LIN {X 0,Y 93.573,Z 328.829,A -85,B 0,C 180,E1 -26788.279,E2 -26788.279} C_VEL
LIN {X 0,Y 93.645,Z 328.819,A -85,B 0,C 180,E1 -26794.239,E2 -26794.239} C_VEL
LIN {X 0,Y 93.653,Z 328.813,A -85,B 0,C 180,E1 -26797.96,E2 -26797.96} C_VEL
LIN {X 0,Y 94.018,Z 328.769,A -85,B 0,C 180,E1 -26807.039,E2 -26807.039} C_VEL
LIN {X 0,Y 94.131,Z 328.757,A -85,B 0,C 180,E1 -26811.41,E2 -26811.41} C_VEL
LIN {X 0,Y 94.763,Z 328.678,A -85,B 0,C 180,E1 -26819.998,E2 -26819.998} C_VEL
LIN {X 0,Y 94.13,Z 328.757,A -85,B 0,C 180,E1 -26828.586,E2 -26828.586} C_VEL
LIN {X 0,Y 93.956,Z 328.78,A -85,B 0,C 180,E1 -26833.486,E2 -26833.486} C_VEL
LIN {X 0,Y 93.653,Z 328.819,A -85,B 0,C 180,E1 -26842.035,E2 -26842.035} C_VEL
LIN {X 0,Y 93.601,Z 328.819,A -85,B 0,C 180,E1 -26846.774,E2 -26846.774} C_VEL
LIN {X 0,Y 93.584,Z 328.823,A -85,B 0,C 180,E1 -26854.298,E2 -26854.298} C_VEL
LIN {X 0,Y 93.537,Z 328.83,A -85,B 0,C 180,E1 -26862.546,E2 -26862.546} C_VEL
LIN {X 0,Y 93.555,Z 328.831,A -85,B 0,C 180,E1 -26868.692,E2 -26868.692} C_VEL
LIN {X 0,Y 93.602,Z 328.824,A -85,B 0,C 180,E1 -26875.679,E2 -26875.679} C_VEL
LIN {X 0,Y 93.669,Z 328.816,A -85,B 0,C 180,E1 -26884.201,E2 -26884.201} C_VEL
LIN {X 0,Y 93.693,Z 328.81,A -85,B 0,C 180,E1 -26887.967,E2 -26887.967} C_VEL
LIN {X 0,Y 94.082,Z 328.759,A -85,B 0,C 180,E1 -26897.044,E2 -26897.044} C_VEL
LIN {X 0,Y 94.207,Z 328.75,A -85,B 0,C 180,E1 -26901.413,E2 -26901.413} C_VEL
LIN {X 0,Y 94.794,Z 328.676,A -85,B 0,C 180,E1 -26909.993,E2 -26909.993} C_VEL
LIN {X 0,Y 94.21,Z 328.751,A -85,B 0,C 180,E1 -26918.573,E2 -26918.573} C_VEL
LIN {X 0,Y 94.181,Z 328.767,A -85,B 0,C 180,E1 -26921.834,E2 -26921.834} C_VEL
LIN {X 0,Y 95.166,Z 331.672,A -85,B 0,C 180,E1 -26922.521,E2 -26922.521} C_VEL
LIN {X 0,Y 101.569,Z 346.523,A -85,B 0,C 180,E1 -26926.174,E2 -26926.174} C_VEL
LIN {X 0,Y 109.633,Z 368.31,A -85,B 0,C 180,E1 -26930.466,E2 -26930.466} C_VEL
LIN {X 0,Y 110.536,Z 370.99,A -85,B 0,C 180,E1 -26930.925,E2 -26930.925} C_VEL
LIN {X 0,Y 105.93,Z 421.379,A -85,B 0,C 180,E1 -26935.46,E2 -26935.46} C_VEL
LIN {X 0,Y 104.057,Z 435.818,A -85,B 0,C 180,E1 -26937.573,E2 -26937.573} C_VEL
LIN {X 0,Y 101.762,Z 448.826,A -85,B 0,C 180,E1 -26940.316,E2 -26940.316} C_VEL
LIN {X 0,Y 99.25,Z 461.551,A -85,B 0,C 180,E1 -26943.946,E2 -26943.946} C_VEL
LIN {X 0,Y 96.668,Z 473.501,A -85,B 0,C 180,E1 -26948.496,E2 -26948.496} C_VEL
LIN {X 0,Y 94.521,Z 483.813,A -85,B 0,C 180,E1 -26953.539,E2 -26953.539} C_VEL
LIN {X 0,Y 92.739,Z 493.445,A -85,B 0,C 180,E1 -26959.62,E2 -26959.62} C_VEL
LIN {X 0,Y 91.805,Z 500.292,A -85,B 0,C 180,E1 -26964.963,E2 -26964.963} C_VEL
LIN {X 0,Y 91.274,Z 506.901,A -85,B 0,C 180,E1 -26971.276,E2 -26971.276} C_VEL
LIN {X 0,Y 91.876,Z 514.034,A -85,B 0,C 180,E1 -26979.868,E2 -26979.868} C_VEL
LIN {X 0,Y 93.831,Z 518.658,A -85,B 0,C 180,E1 -26987.017,E2 -26987.017} C_VEL
LIN {X 0,Y 95.951,Z 521.091,A -85,B 0,C 180,E1 -26991.578,E2 -26991.578} C_VEL
LIN {X 0,Y 98.609,Z 523.092,A -85,B 0,C 180,E1 -26996.015,E2 -26996.015} C_VEL
LIN {X 0,Y 101.749,Z 524.592,A -85,B 0,C 180,E1 -27000.002,E2 -27000.002} C_VEL
LIN {X 0,Y 105.656,Z 525.69,A -85,B 0,C 180,E1 -27004.008,E2 -27004.008} C_VEL
LIN {X 0,Y 109.634,Z 526.281,A -85,B 0,C 180,E1 -27007.368,E2 -27007.368} C_VEL
LIN {X 0,Y 114.426,Z 526.503,A -85,B 0,C 180,E1 -27010.73,E2 -27010.73} C_VEL
LIN {X 0,Y 119.307,Z 526.284,A -85,B 0,C 180,E1 -27013.63,E2 -27013.63} C_VEL
LIN {X 0,Y 124.666,Z 525.596,A -85,B 0,C 180,E1 -27016.374,E2 -27016.374} C_VEL
LIN {X 0,Y 135.294,Z 523.2,A -85,B 0,C 180,E1 -27020.795,E2 -27020.795} C_VEL
LIN {X 0,Y 146.652,Z 519.189,A -85,B 0,C 180,E1 -27024.444,E2 -27024.444} C_VEL
LIN {X 0,Y 158.313,Z 513.62,A -85,B 0,C 180,E1 -27027.414,E2 -27027.414} C_VEL
LIN {X 0,Y 167.136,Z 508.313,A -85,B 0,C 180,E1 -27029.296,E2 -27029.296} C_VEL
LIN {X 0,Y 165.242,Z 509.715,A -85,B 0,C 180,E1 -27030.279,E2 -27030.279} C_VEL
LIN {X 0,Y 154.143,Z 516.659,A -85,B 0,C 180,E1 -27032.507,E2 -27032.507} C_VEL
LIN {X 0,Y 145.218,Z 521.23,A -85,B 0,C 180,E1 -27034.657,E2 -27034.657} C_VEL
LIN {X 0,Y 133.848,Z 525.943,A -85,B 0,C 180,E1 -27038.053,E2 -27038.053} C_VEL
LIN {X 0,Y 123.437,Z 529.163,A -85,B 0,C 180,E1 -27042.268,E2 -27042.268} C_VEL
LIN {X 0,Y 114.003,Z 531.067,A -85,B 0,C 180,E1 -27047.316,E2 -27047.316} C_VEL
LIN {X 0,Y 106.022,Z 531.693,A -85,B 0,C 180,E1 -27053.386,E2 -27053.386} C_VEL
LIN {X 0,Y 99.465,Z 530.999,A -85,B 0,C 180,E1 -27060.367,E2 -27060.367} C_VEL
LIN {X 0,Y 94.915,Z 528.991,A -85,B 0,C 180,E1 -27068.28,E2 -27068.28} C_VEL
LIN {X 0,Y 92.801,Z 525.673,A -85,B 0,C 180,E1 -27076.876,E2 -27076.876} C_VEL
LIN {X 0,Y 92.558,Z 522.492,A -85,B 0,C 180,E1 -27082.906,E2 -27082.906} C_VEL
LIN {X 0,Y 92.895,Z 519.232,A -85,B 0,C 180,E1 -27087.839,E2 -27087.839} C_VEL
LIN {X 0,Y 92.777,Z 514.534,A -85,B 0,C 180,E1 -27093.264,E2 -27093.264} C_VEL
LIN {X 0,Y 92.839,Z 508.649,A -85,B 0,C 180,E1 -27098.714,E2 -27098.714} C_VEL
LIN {X 0,Y 93.733,Z 499.874,A -85,B 0,C 180,E1 -27105.22,E2 -27105.22} C_VEL
LIN {X 0,Y 95.279,Z 490.866,A -85,B 0,C 180,E1 -27110.515,E2 -27110.515} C_VEL
LIN {X 0,Y 97.615,Z 479.729,A -85,B 0,C 180,E1 -27115.598,E2 -27115.598} C_VEL
LIN {X 0,Y 99.953,Z 468.688,A -85,B 0,C 180,E1 -27119.489,E2 -27119.489} C_VEL
LIN {X 0,Y 102.558,Z 455.448,A -85,B 0,C 180,E1 -27122.955,E2 -27122.955} C_VEL
LIN {X 0,Y 104.664,Z 442.605,A -85,B 0,C 180,E1 -27125.394,E2 -27125.394} C_VEL
LIN {X 0,Y 106.08,Z 430.388,A -85,B 0,C 180,E1 -27127.008,E2 -27127.008} C_VEL
LIN {X 0,Y 109.326,Z 392.754,A -85,B 0,C 180,E1 -27130.449,E2 -27130.449} C_VEL
LIN {X 0,Y 107.869,Z 369.994,A -85,B 0,C 180,E1 -27133.101,E2 -27133.101} C_VEL
LIN {X 0,Y 107.342,Z 367.864,A -85,B 0,C 180,E1 -27133.437,E2 -27133.437} C_VEL
LIN {X 0,Y 105.36,Z 362.63,A -85,B 0,C 180,E1 -27134.438,E2 -27134.438} C_VEL
LIN {X 0,Y 100.496,Z 354.863,A -85,B 0,C 180,E1 -27136.508,E2 -27136.508} C_VEL
LIN {X 0,Y 96.186,Z 348.926,A -85,B 0,C 180,E1 -27138.421,E2 -27138.421} C_VEL
LIN {X 0,Y 92.4,Z 342.627,A -85,B 0,C 180,E1 -27140.358,E2 -27140.358} C_VEL
LIN {X 0,Y 87.501,Z 332.578,A -85,B 0,C 180,E1 -27143.394,E2 -27143.394} C_VEL
LIN {X 0,Y 86.506,Z 329.708,A -85,B 0,C 180,E1 -27144.339,E2 -27144.339} C_VEL
LIN {X 0,Y 86.567,Z 329.702,A -85,B 0,C 180,E1 -27153.263,E2 -27153.263} C_VEL
LIN {X 0,Y 86.598,Z 329.698,A -85,B 0,C 180,E1 -27161.055,E2 -27161.055} C_VEL
LIN {X 0,Y 86.861,Z 329.658,A -85,B 0,C 180,E1 -27166.158,E2 -27166.158} C_VEL
LIN {X 0,Y 87.026,Z 329.644,A -85,B 0,C 180,E1 -27170.703,E2 -27170.703} C_VEL
LIN {X 0,Y 87.693,Z 329.559,A -85,B 0,C 180,E1 -27179.998,E2 -27179.998} C_VEL
LIN {X 0,Y 87.024,Z 329.639,A -85,B 0,C 180,E1 -27189.293,E2 -27189.293} C_VEL
LIN {X 0,Y 86.86,Z 329.666,A -85,B 0,C 180,E1 -27194.046,E2 -27194.046} C_VEL
LIN {X 0,Y 86.597,Z 329.69,A -85,B 0,C 180,E1 -27198.941,E2 -27198.941} C_VEL
LIN {X 0,Y 86.566,Z 329.695,A -85,B 0,C 180,E1 -27206.736,E2 -27206.736} C_VEL
LIN {X 0,Y 86.504,Z 329.702,A -85,B 0,C 180,E1 -27215.659,E2 -27215.659} C_VEL
LIN {X 0,Y 86.48,Z 329.708,A -85,B 0,C 180,E1 -27222.991,E2 -27222.991} C_VEL
LIN {X 0,Y 86.475,Z 329.713,A -85,B 0,C 180,E1 -27229.44,E2 -27229.44} C_VEL
LIN {X 0,Y 86.547,Z 329.703,A -85,B 0,C 180,E1 -27235.354,E2 -27235.354} C_VEL
LIN {X 0,Y 86.584,Z 329.697,A -85,B 0,C 180,E1 -27243.231,E2 -27243.231} C_VEL
LIN {X 0,Y 86.646,Z 329.687,A -85,B 0,C 180,E1 -27251.062,E2 -27251.062} C_VEL
LIN {X 0,Y 86.95,Z 329.651,A -85,B 0,C 180,E1 -27255.961,E2 -27255.961} C_VEL
LIN {X 0,Y 87.111,Z 329.633,A -85,B 0,C 180,E1 -27260.708,E2 -27260.708} C_VEL
LIN {X 0,Y 87.722,Z 329.558,A -85,B 0,C 180,E1 -27269.993,E2 -27269.993} C_VEL
LIN {X 0,Y 87.135,Z 329.63,A -85,B 0,C 180,E1 -27279.421,E2 -27279.421} C_VEL
LIN {X 0,Y 88.182,Z 332.606,A -85,B 0,C 180,E1 -27280.249,E2 -27280.249} C_VEL
LIN {X 0,Y 94.846,Z 347.726,A -85,B 0,C 180,E1 -27284.444,E2 -27284.444} C_VEL
LIN {X 0,Y 102.434,Z 368.321,A -85,B 0,C 180,E1 -27288.89,E2 -27288.89} C_VEL
LIN {X 0,Y 103.782,Z 372.236,A -85,B 0,C 180,E1 -27289.638,E2 -27289.638} C_VEL
LIN {X 0,Y 99.129,Z 421.425,A -85,B 0,C 180,E1 -27294.314,E2 -27294.314} C_VEL
LIN {X 0,Y 97.199,Z 435.818,A -85,B 0,C 180,E1 -27296.53,E2 -27296.53} C_VEL
LIN {X 0,Y 94.953,Z 448.117,A -85,B 0,C 180,E1 -27299.226,E2 -27299.226} C_VEL
LIN {X 0,Y 92.302,Z 461.049,A -85,B 0,C 180,E1 -27303.121,E2 -27303.121} C_VEL
LIN {X 0,Y 89.803,Z 472.245,A -85,B 0,C 180,E1 -27307.595,E2 -27307.595} C_VEL
LIN {X 0,Y 87.602,Z 482.61,A -85,B 0,C 180,E1 -27312.944,E2 -27312.944} C_VEL
LIN {X 0,Y 85.789,Z 491.966,A -85,B 0,C 180,E1 -27319.055,E2 -27319.055} C_VEL
LIN {X 0,Y 84.854,Z 498.799,A -85,B 0,C 180,E1 -27324.568,E2 -27324.568} C_VEL
LIN {X 0,Y 84.283,Z 505.708,A -85,B 0,C 180,E1 -27331.352,E2 -27331.352} C_VEL
LIN {X 0,Y 84.613,Z 511.599,A -85,B 0,C 180,E1 -27338.541,E2 -27338.541} C_VEL
LIN {X 0,Y 86.562,Z 517.223,A -85,B 0,C 180,E1 -27346.919,E2 -27346.919} C_VEL
LIN {X 0,Y 90.737,Z 521.822,A -85,B 0,C 180,E1 -27355.56,E2 -27355.56} C_VEL
LIN {X 0,Y 93.852,Z 523.72,A -85,B 0,C 180,E1 -27360.002,E2 -27360.002} C_VEL
LIN {X 0,Y 98.798,Z 525.543,A -85,B 0,C 180,E1 -27365.331,E2 -27365.331} C_VEL
LIN {X 0,Y 107.894,Z 526.949,A -85,B 0,C 180,E1 -27372.349,E2 -27372.349} C_VEL
LIN {X 0,Y 118.23,Z 526.65,A -85,B 0,C 180,E1 -27378.029,E2 -27378.029} C_VEL
LIN {X 0,Y 129.371,Z 524.824,A -85,B 0,C 180,E1 -27382.582,E2 -27382.582} C_VEL
LIN {X 0,Y 135.32,Z 523.307,A -85,B 0,C 180,E1 -27384.552,E2 -27384.552} C_VEL
LIN {X 0,Y 145.313,Z 519.918,A -85,B 0,C 180,E1 -27387.354,E2 -27387.354} C_VEL
LIN {X 0,Y 152.834,Z 516.661,A -85,B 0,C 180,E1 -27389.127,E2 -27389.127} C_VEL
LIN {X 0,Y 153.61,Z 516.346,A -85,B 0,C 180,E1 -27389.642,E2 -27389.642} C_VEL
LIN {X 0,Y 144.329,Z 520.911,A -85,B 0,C 180,E1 -27391.572,E2 -27391.572} C_VEL
LIN {X 0,Y 135.409,Z 524.497,A -85,B 0,C 180,E1 -27393.874,E2 -27393.874} C_VEL
LIN {X 0,Y 129.616,Z 526.446,A -85,B 0,C 180,E1 -27395.595,E2 -27395.595} C_VEL
LIN {X 0,Y 118.788,Z 529.296,A -85,B 0,C 180,E1 -27399.739,E2 -27399.739} C_VEL
LIN {X 0,Y 108.887,Z 530.811,A -85,B 0,C 180,E1 -27404.781,E2 -27404.781} C_VEL
LIN {X 0,Y 100.416,Z 531.081,A -85,B 0,C 180,E1 -27410.97,E2 -27410.97} C_VEL
LIN {X 0,Y 93.38,Z 530.082,A -85,B 0,C 180,E1 -27418.22,E2 -27418.22} C_VEL
LIN {X 0,Y 88.425,Z 527.802,A -85,B 0,C 180,E1 -27426.595,E2 -27426.595} C_VEL
LIN {X 0,Y 86.034,Z 524.174,A -85,B 0,C 180,E1 -27435.823,E2 -27435.823} C_VEL
LIN {X 0,Y 85.757,Z 520.047,A -85,B 0,C 180,E1 -27443.597,E2 -27443.597} C_VEL
LIN {X 0,Y 86.024,Z 517.323,A -85,B 0,C 180,E1 -27447.667,E2 -27447.667} C_VEL
LIN {X 0,Y 85.863,Z 512.343,A -85,B 0,C 180,E1 -27453.527,E2 -27453.527} C_VEL
LIN {X 0,Y 86.057,Z 504.633,A -85,B 0,C 180,E1 -27460.654,E2 -27460.654} C_VEL
LIN {X 0,Y 87.377,Z 495.19,A -85,B 0,C 180,E1 -27467.561,E2 -27467.561} C_VEL
LIN {X 0,Y 89.255,Z 485.216,A -85,B 0,C 180,E1 -27473.191,E2 -27473.191} C_VEL
LIN {X 0,Y 91.665,Z 474.119,A -85,B 0,C 180,E1 -27478.014,E2 -27478.014} C_VEL
LIN {X 0,Y 93.944,Z 463.458,A -85,B 0,C 180,E1 -27481.583,E2 -27481.583} C_VEL
LIN {X 0,Y 96.379,Z 450.858,A -85,B 0,C 180,E1 -27484.733,E2 -27484.733} C_VEL
LIN {X 0,Y 98.532,Z 437.173,A -85,B 0,C 180,E1 -27487.165,E2 -27487.165} C_VEL
LIN {X 0,Y 100.132,Z 420.928,A -85,B 0,C 180,E1 -27489.016,E2 -27489.016} C_VEL
LIN {X 0,Y 102.571,Z 392.894,A -85,B 0,C 180,E1 -27491.696,E2 -27491.696} C_VEL
LIN {X 0,Y 101.351,Z 371.639,A -85,B 0,C 180,E1 -27494.346,E2 -27494.346} C_VEL
LIN {X 0,Y 95.522,Z 351.056,A -85,B 0,C 180,E1 -27498.356,E2 -27498.356} C_VEL
LIN {X 0,Y 93.12,Z 344.081,A -85,B 0,C 180,E1 -27499.948,E2 -27499.948} C_VEL
LIN {X 0,Y 92.4,Z 342.627,A -85,B 0,C 180,E1 -27500.358,E2 -27500.358} C_VEL
LIN {X 0,Y 89.675,Z 338.423,A -85,B 0,C 180,E1 -27502.024,E2 -27502.024} C_VEL
LIN {X 0,Y 86.516,Z 335.212,A -85,B 0,C 180,E1 -27504.303,E2 -27504.303} C_VEL
LIN {X 0,Y 84.439,Z 333.568,A -85,B 0,C 180,E1 -27506.148,E2 -27506.148} C_VEL
LIN {X 0,Y 81.696,Z 331.776,A -85,B 0,C 180,E1 -27509.405,E2 -27509.405} C_VEL
LIN {X 0,Y 79.855,Z 330.78,A -85,B 0,C 180,E1 -27513.182,E2 -27513.182} C_VEL
LIN {X 0,Y 79.409,Z 330.581,A -85,B 0,C 180,E1 -27515.896,E2 -27515.896} C_VEL
LIN {X 0,Y 79.69,Z 330.551,A -85,B 0,C 180,E1 -27524.656,E2 -27524.656} C_VEL
LIN {X 0,Y 79.91,Z 330.531,A -85,B 0,C 180,E1 -27529.867,E2 -27529.867} C_VEL
LIN {X 0,Y 80.622,Z 330.44,A -85,B 0,C 180,E1 -27539.998,E2 -27539.998} C_VEL
LIN {X 0,Y 79.909,Z 330.523,A -85,B 0,C 180,E1 -27550.128,E2 -27550.128} C_VEL
LIN {X 0,Y 79.688,Z 330.559,A -85,B 0,C 180,E1 -27555.339,E2 -27555.339} C_VEL
LIN {X 0,Y 79.476,Z 330.581,A -85,B 0,C 180,E1 -27560.712,E2 -27560.712} C_VEL
LIN {X 0,Y 79.468,Z 330.578,A -85,B 0,C 180,E1 -27567.818,E2 -27567.818} C_VEL
LIN {X 0,Y 79.372,Z 330.598,A -85,B 0,C 180,E1 -27572.088,E2 -27572.088} C_VEL
LIN {X 0,Y 79.365,Z 330.597,A -85,B 0,C 180,E1 -27578.303,E2 -27578.303} C_VEL
LIN {X 0,Y 79.412,Z 330.586,A -85,B 0,C 180,E1 -27585.069,E2 -27585.069} C_VEL
LIN {X 0,Y 79.399,Z 330.586,A -85,B 0,C 180,E1 -27592.806,E2 -27592.806} C_VEL
LIN {X 0,Y 79.386,Z 330.596,A -85,B 0,C 180,E1 -27597.909,E2 -27597.909} C_VEL
LIN {X 0,Y 79.525,Z 330.577,A -85,B 0,C 180,E1 -27603.77,E2 -27603.77} C_VEL
LIN {X 0,Y 79.513,Z 330.572,A -85,B 0,C 180,E1 -27609.289,E2 -27609.289} C_VEL
LIN {X 0,Y 79.838,Z 330.538,A -85,B 0,C 180,E1 -27615.526,E2 -27615.526} C_VEL
LIN {X 0,Y 79.991,Z 330.518,A -85,B 0,C 180,E1 -27619.872,E2 -27619.872} C_VEL
LIN {X 0,Y 80.65,Z 330.439,A -85,B 0,C 180,E1 -27629.992,E2 -27629.992} C_VEL
LIN {X 0,Y 80.082,Z 330.514,A -85,B 0,C 180,E1 -27636.606,E2 -27636.606} C_VEL
LIN {X 0,Y 81.156,Z 333.469,A -85,B 0,C 180,E1 -27637.533,E2 -27637.533} C_VEL
LIN {X 0,Y 84.237,Z 339.738,A -85,B 0,C 180,E1 -27639.747,E2 -27639.747} C_VEL
LIN {X 0,Y 89.836,Z 353.407,A -85,B 0,C 180,E1 -27643.654,E2 -27643.654} C_VEL
LIN {X 0,Y 96.539,Z 371.954,A -85,B 0,C 180,E1 -27647.861,E2 -27647.861} C_VEL
LIN {X 0,Y 97.091,Z 374.405,A -85,B 0,C 180,E1 -27648.287,E2 -27648.287} C_VEL
LIN {X 0,Y 92.273,Z 422.261,A -85,B 0,C 180,E1 -27653.172,E2 -27653.172} C_VEL
LIN {X 0,Y 90.132,Z 436.987,A -85,B 0,C 180,E1 -27655.639,E2 -27655.639} C_VEL
LIN {X 0,Y 87.69,Z 449.666,A -85,B 0,C 180,E1 -27658.731,E2 -27658.731} C_VEL
LIN {X 0,Y 84.893,Z 462.653,A -85,B 0,C 180,E1 -27663.053,E2 -27663.053} C_VEL
LIN {X 0,Y 82.253,Z 474.252,A -85,B 0,C 180,E1 -27668.264,E2 -27668.264} C_VEL
LIN {X 0,Y 80.132,Z 483.916,A -85,B 0,C 180,E1 -27673.837,E2 -27673.837} C_VEL
LIN {X 0,Y 78.624,Z 491.944,A -85,B 0,C 180,E1 -27679.608,E2 -27679.608} C_VEL
LIN {X 0,Y 77.569,Z 500.264,A -85,B 0,C 180,E1 -27687.073,E2 -27687.073} C_VEL
LIN {X 0,Y 77.327,Z 507.531,A -85,B 0,C 180,E1 -27695.317,E2 -27695.317} C_VEL
LIN {X 0,Y 78.687,Z 514.056,A -85,B 0,C 180,E1 -27704.46,E2 -27704.46} C_VEL
LIN {X 0,Y 81.576,Z 518.831,A -85,B 0,C 180,E1 -27712.577,E2 -27712.577} C_VEL
LIN {X 0,Y 85.984,Z 522.477,A -85,B 0,C 180,E1 -27720.002,E2 -27720.002} C_VEL
LIN {X 0,Y 92.002,Z 525.211,A -85,B 0,C 180,E1 -27726.858,E2 -27726.858} C_VEL
LIN {X 0,Y 101.475,Z 527.183,A -85,B 0,C 180,E1 -27734.208,E2 -27734.208} C_VEL
LIN {X 0,Y 112.153,Z 527.456,A -85,B 0,C 180,E1 -27739.987,E2 -27739.987} C_VEL
LIN {X 0,Y 123.603,Z 526.25,A -85,B 0,C 180,E1 -27744.554,E2 -27744.554} C_VEL
LIN {X 0,Y 135.477,Z 523.546,A -85,B 0,C 180,E1 -27748.149,E2 -27748.149} C_VEL
LIN {X 0,Y 138.821,Z 522.561,A -85,B 0,C 180,E1 -27749.023,E2 -27749.023} C_VEL
LIN {X 0,Y 137.697,Z 523.035,A -85,B 0,C 180,E1 -27749.831,E2 -27749.831} C_VEL
LIN {X 0,Y 125.623,Z 526.855,A -85,B 0,C 180,E1 -27752.965,E2 -27752.965} C_VEL
LIN {X 0,Y 114.378,Z 529.299,A -85,B 0,C 180,E1 -27757.003,E2 -27757.003} C_VEL
LIN {X 0,Y 104.02,Z 530.489,A -85,B 0,C 180,E1 -27762.01,E2 -27762.01} C_VEL
LIN {X 0,Y 95.011,Z 530.427,A -85,B 0,C 180,E1 -27768.276,E2 -27768.276} C_VEL
LIN {X 0,Y 87.46,Z 529.073,A -85,B 0,C 180,E1 -27775.784,E2 -27775.784} C_VEL
LIN {X 0,Y 82.043,Z 526.479,A -85,B 0,C 180,E1 -27784.651,E2 -27784.651} C_VEL
LIN {X 0,Y 79.333,Z 522.546,A -85,B 0,C 180,E1 -27794.597,E2 -27794.597} C_VEL
LIN {X 0,Y 78.937,Z 518.578,A -85,B 0,C 180,E1 -27802.334,E2 -27802.334} C_VEL
LIN {X 0,Y 79.172,Z 515.331,A -85,B 0,C 180,E1 -27807.465,E2 -27807.465} C_VEL
LIN {X 0,Y 78.966,Z 509.994,A -85,B 0,C 180,E1 -27813.835,E2 -27813.835} C_VEL
LIN {X 0,Y 79.247,Z 501.612,A -85,B 0,C 180,E1 -27821.793,E2 -27821.793} C_VEL
LIN {X 0,Y 80.764,Z 491.781,A -85,B 0,C 180,E1 -27829.052,E2 -27829.052} C_VEL
LIN {X 0,Y 82.905,Z 481.221,A -85,B 0,C 180,E1 -27835.084,E2 -27835.084} C_VEL
LIN {X 0,Y 85.595,Z 469.314,A -85,B 0,C 180,E1 -27840.198,E2 -27840.198} C_VEL
LIN {X 0,Y 88.112,Z 457.694,A -85,B 0,C 180,E1 -27843.946,E2 -27843.946} C_VEL
LIN {X 0,Y 90.533,Z 444.586,A -85,B 0,C 180,E1 -27846.991,E2 -27846.991} C_VEL
LIN {X 0,Y 92.221,Z 432.548,A -85,B 0,C 180,E1 -27848.96,E2 -27848.96} C_VEL
LIN {X 0,Y 95.931,Z 394.052,A -85,B 0,C 180,E1 -27852.985,E2 -27852.985} C_VEL
LIN {X 0,Y 94.901,Z 373.415,A -85,B 0,C 180,E1 -27855.751,E2 -27855.751} C_VEL
LIN {X 0,Y 89.374,Z 353.596,A -85,B 0,C 180,E1 -27859.863,E2 -27859.863} C_VEL
LIN {X 0,Y 87.144,Z 347.089,A -85,B 0,C 180,E1 -27861.494,E2 -27861.494} C_VEL
LIN {X 0,Y 81.935,Z 336.258,A -85,B 0,C 180,E1 -27865.085,E2 -27865.085} C_VEL
LIN {X 0,Y 79.562,Z 331.488,A -85,B 0,C 180,E1 -27866.865,E2 -27866.865} C_VEL
LIN {X 0,Y 79.395,Z 330.594,A -85,B 0,C 180,E1 -27867.165,E2 -27867.165} C_VEL
LIN {X 0,Y 79.508,Z 330.58,A -85,B 0,C 180,E1 -27873.768,E2 -27873.768} C_VEL
LIN {X 0,Y 79.409,Z 330.581,A -85,B 0,C 180,E1 -27875.896,E2 -27875.896} C_VEL
LIN {X 0,Y 78.681,Z 330.683,A -85,B 0,C 180,E1 -27880.134,E2 -27880.134} C_VEL
LIN {X 0,Y 77.128,Z 330.878,A -85,B 0,C 180,E1 -27884.358,E2 -27884.358} C_VEL
LIN {X 0,Y 73.356,Z 331.346,A -85,B 0,C 180,E1 -27896.354,E2 -27896.354} C_VEL
LIN {X 0,Y 73.472,Z 331.326,A -85,B 0,C 180,E1 -27899.511,E2 -27899.511} C_VEL
LIN {X 0,Y 72.916,Z 331.395,A -85,B 0,C 180,E1 -27906.381,E2 -27906.381} C_VEL
LIN {X 0,Y 72.809,Z 331.407,A -85,B 0,C 180,E1 -27911.128,E2 -27911.128} C_VEL
LIN {X 0,Y 72.506,Z 331.45,A -85,B 0,C 180,E1 -27916.902,E2 -27916.902} C_VEL
LIN {X 0,Y 72.367,Z 331.47,A -85,B 0,C 180,E1 -27922.856,E2 -27922.856} C_VEL
LIN {X 0,Y 72.36,Z 331.466,A -85,B 0,C 180,E1 -27929.05,E2 -27929.05} C_VEL
LIN {X 0,Y 72.292,Z 331.472,A -85,B 0,C 180,E1 -27935.68,E2 -27935.68} C_VEL
LIN {X 0,Y 72.261,Z 331.478,A -85,B 0,C 180,E1 -27942.903,E2 -27942.903} C_VEL
LIN {X 0,Y 72.306,Z 331.474,A -85,B 0,C 180,E1 -27951.036,E2 -27951.036} C_VEL
LIN {X 0,Y 72.304,Z 331.473,A -85,B 0,C 180,E1 -27954.317,E2 -27954.317} C_VEL
LIN {X 0,Y 72.376,Z 331.461,A -85,B 0,C 180,E1 -27960.946,E2 -27960.946} C_VEL
LIN {X 0,Y 72.394,Z 331.465,A -85,B 0,C 180,E1 -27967.143,E2 -27967.143} C_VEL
LIN {X 0,Y 72.755,Z 331.421,A -85,B 0,C 180,E1 -27975.002,E2 -27975.002} C_VEL
LIN {X 0,Y 72.878,Z 331.4,A -85,B 0,C 180,E1 -27978.872,E2 -27978.872} C_VEL
LIN {X 0,Y 73.577,Z 331.32,A -85,B 0,C 180,E1 -27989.991,E2 -27989.991} C_VEL
LIN {X 0,Y 73.219,Z 331.359,A -85,B 0,C 180,E1 -27993.258,E2 -27993.258} C_VEL
LIN {X 0,Y 74.182,Z 334.307,A -85,B 0,C 180,E1 -27994.406,E2 -27994.406} C_VEL
LIN {X 0,Y 78.483,Z 342.94,A -85,B 0,C 180,E1 -27997.882,E2 -27997.882} C_VEL
LIN {X 0,Y 84.157,Z 357.131,A -85,B 0,C 180,E1 -28002.255,E2 -28002.255} C_VEL
LIN {X 0,Y 90.319,Z 374.686,A -85,B 0,C 180,E1 -28006.596,E2 -28006.596} C_VEL
LIN {X 0,Y 85.443,Z 422.933,A -85,B 0,C 180,E1 -28011.893,E2 -28011.893} C_VEL
LIN {X 0,Y 83.187,Z 437.447,A -85,B 0,C 180,E1 -28014.493,E2 -28014.493} C_VEL
LIN {X 0,Y 80.496,Z 450.947,A -85,B 0,C 180,E1 -28018.078,E2 -28018.078} C_VEL
LIN {X 0,Y 77.779,Z 462.885,A -85,B 0,C 180,E1 -28022.405,E2 -28022.405} C_VEL
LIN {X 0,Y 74.967,Z 474.83,A -85,B 0,C 180,E1 -28028.27,E2 -28028.27} C_VEL
LIN {X 0,Y 72.769,Z 484.728,A -85,B 0,C 180,E1 -28034.651,E2 -28034.651} C_VEL
LIN {X 0,Y 71.202,Z 493.839,A -85,B 0,C 180,E1 -28042.13,E2 -28042.13} C_VEL
LIN {X 0,Y 70.429,Z 501.536,A -85,B 0,C 180,E1 -28050.073,E2 -28050.073} C_VEL
LIN {X 0,Y 70.705,Z 508.983,A -85,B 0,C 180,E1 -28059.644,E2 -28059.644} C_VEL
LIN {X 0,Y 72.767,Z 514.871,A -85,B 0,C 180,E1 -28068.865,E2 -28068.865} C_VEL
LIN {X 0,Y 77.311,Z 520.21,A -85,B 0,C 180,E1 -28078.619,E2 -28078.619} C_VEL
LIN {X 0,Y 81.843,Z 523.141,A -85,B 0,C 180,E1 -28084.929,E2 -28084.929} C_VEL
LIN {X 0,Y 86.119,Z 524.977,A -85,B 0,C 180,E1 -28089.396,E2 -28089.396} C_VEL
LIN {X 0,Y 95.175,Z 527.199,A -85,B 0,C 180,E1 -28096.314,E2 -28096.314} C_VEL
LIN {X 0,Y 106.253,Z 528.059,A -85,B 0,C 180,E1 -28102.209,E2 -28102.209} C_VEL
LIN {X 0,Y 118.057,Z 527.436,A -85,B 0,C 180,E1 -28106.776,E2 -28106.776} C_VEL
LIN {X 0,Y 124.606,Z 526.461,A -85,B 0,C 180,E1 -28108.795,E2 -28108.795} C_VEL
LIN {X 0,Y 123.272,Z 526.883,A -85,B 0,C 180,E1 -28109.813,E2 -28109.813} C_VEL
LIN {X 0,Y 110.256,Z 529.223,A -85,B 0,C 180,E1 -28114.059,E2 -28114.059} C_VEL
LIN {X 0,Y 99.411,Z 530.023,A -85,B 0,C 180,E1 -28118.97,E2 -28118.97} C_VEL
LIN {X 0,Y 89.845,Z 529.619,A -85,B 0,C 180,E1 -28125.266,E2 -28125.266} C_VEL
LIN {X 0,Y 81.732,Z 527.988,A -85,B 0,C 180,E1 -28133.007,E2 -28133.007} C_VEL
LIN {X 0,Y 75.797,Z 525.061,A -85,B 0,C 180,E1 -28142.393,E2 -28142.393} C_VEL
LIN {X 0,Y 72.702,Z 520.826,A -85,B 0,C 180,E1 -28153.153,E2 -28153.153} C_VEL
LIN {X 0,Y 72.366,Z 514.983,A -85,B 0,C 180,E1 -28164.436,E2 -28164.436} C_VEL
LIN {X 0,Y 72.226,Z 511.047,A -85,B 0,C 180,E1 -28170.009,E2 -28170.009} C_VEL
LIN {X 0,Y 72.039,Z 504.91,A -85,B 0,C 180,E1 -28177.013,E2 -28177.013} C_VEL
LIN {X 0,Y 72.859,Z 495.797,A -85,B 0,C 180,E1 -28185.28,E2 -28185.28} C_VEL
LIN {X 0,Y 74.603,Z 486.121,A -85,B 0,C 180,E1 -28192.144,E2 -28192.144} C_VEL
LIN {X 0,Y 76.997,Z 475.592,A -85,B 0,C 180,E1 -28197.898,E2 -28197.898} C_VEL
LIN {X 0,Y 79.67,Z 463.896,A -85,B 0,C 180,E1 -28202.71,E2 -28202.71} C_VEL
LIN {X 0,Y 82.233,Z 451.901,A -85,B 0,C 180,E1 -28206.369,E2 -28206.369} C_VEL
LIN {X 0,Y 84.642,Z 438.246,A -85,B 0,C 180,E1 -28209.286,E2 -28209.286} C_VEL
LIN {X 0,Y 86.259,Z 424.458,A -85,B 0,C 180,E1 -28211.26,E2 -28211.26} C_VEL
LIN {X 0,Y 89.228,Z 393.764,A -85,B 0,C 180,E1 -28214.608,E2 -28214.608} C_VEL
LIN {X 0,Y 88.341,Z 374.688,A -85,B 0,C 180,E1 -28217.351,E2 -28217.351} C_VEL
LIN {X 0,Y 82.585,Z 353.674,A -85,B 0,C 180,E1 -28222.2,E2 -28222.2} C_VEL
LIN {X 0,Y 78.483,Z 343.957,A -85,B 0,C 180,E1 -28225.385,E2 -28225.385} C_VEL
LIN {X 0,Y 73.68,Z 334.843,A -85,B 0,C 180,E1 -28229.152,E2 -28229.152} C_VEL
LIN {X 0,Y 72.51,Z 332.392,A -85,B 0,C 180,E1 -28230.213,E2 -28230.213} C_VEL
LIN {X 0,Y 72.34,Z 331.473,A -85,B 0,C 180,E1 -28230.536,E2 -28230.536} C_VEL
LIN {X 0,Y 72.369,Z 331.462,A -85,B 0,C 180,E1 -28237.139,E2 -28237.139} C_VEL
LIN {X 0,Y 72.68,Z 331.423,A -85,B 0,C 180,E1 -28245.246,E2 -28245.246} C_VEL
LIN {X 0,Y 72.81,Z 331.415,A -85,B 0,C 180,E1 -28248.866,E2 -28248.866} C_VEL
LIN {X 0,Y 73.472,Z 331.326,A -85,B 0,C 180,E1 -28259.511,E2 -28259.511} C_VEL
LIN {X 0,Y 73.413,Z 331.347,A -85,B 0,C 180,E1 -28262.522,E2 -28262.522} C_VEL
LIN {X 0,Y 71.964,Z 331.527,A -85,B 0,C 180,E1 -28267.002,E2 -28267.002} C_VEL
LIN {X 0,Y 69.692,Z 331.796,A -85,B 0,C 180,E1 -28271.467,E2 -28271.467} C_VEL
LIN {X 0,Y 65.498,Z 332.324,A -85,B 0,C 180,E1 -28281.55,E2 -28281.55} C_VEL
LIN {X 0,Y 65.202,Z 332.356,A -85,B 0,C 180,E1 -28285.203,E2 -28285.203} C_VEL
LIN {X 0,Y 65.171,Z 332.366,A -85,B 0,C 180,E1 -28292.625,E2 -28292.625} C_VEL
LIN {X 0,Y 65.191,Z 332.364,A -85,B 0,C 180,E1 -28300.998,E2 -28300.998} C_VEL
LIN {X 0,Y 65.216,Z 332.36,A -85,B 0,C 180,E1 -28309.707,E2 -28309.707} C_VEL
LIN {X 0,Y 65.256,Z 332.351,A -85,B 0,C 180,E1 -28319.489,E2 -28319.489} C_VEL
LIN {X 0,Y 65.239,Z 332.358,A -85,B 0,C 180,E1 -28324.467,E2 -28324.467} C_VEL
LIN {X 0,Y 65.649,Z 332.307,A -85,B 0,C 180,E1 -28334.457,E2 -28334.457} C_VEL
LIN {X 0,Y 65.778,Z 332.283,A -85,B 0,C 180,E1 -28337.653,E2 -28337.653} C_VEL
LIN {X 0,Y 66.414,Z 332.32,A -85,B 0,C 180,E1 -28349.422,E2 -28349.422} C_VEL
LIN {X 0,Y 67.832,Z 335.69,A -85,B 0,C 180,E1 -28351.01,E2 -28351.01} C_VEL
LIN {X 0,Y 73.112,Z 347.039,A -85,B 0,C 180,E1 -28356.09,E2 -28356.09} C_VEL
LIN {X 0,Y 77.966,Z 359.468,A -85,B 0,C 180,E1 -28360.287,E2 -28360.287} C_VEL
LIN {X 0,Y 83.76,Z 376.151,A -85,B 0,C 180,E1 -28364.844,E2 -28364.844} C_VEL
LIN {X 0,Y 78.604,Z 423.608,A -85,B 0,C 180,E1 -28370.379,E2 -28370.379} C_VEL
LIN {X 0,Y 76.36,Z 437.382,A -85,B 0,C 180,E1 -28373.025,E2 -28373.025} C_VEL
LIN {X 0,Y 73.72,Z 450.181,A -85,B 0,C 180,E1 -28376.657,E2 -28376.657} C_VEL
LIN {X 0,Y 70.865,Z 462.19,A -85,B 0,C 180,E1 -28381.332,E2 -28381.332} C_VEL
LIN {X 0,Y 68.081,Z 473.541,A -85,B 0,C 180,E1 -28387.281,E2 -28387.281} C_VEL
LIN {X 0,Y 65.62,Z 484.345,A -85,B 0,C 180,E1 -28394.806,E2 -28394.806} C_VEL
LIN {X 0,Y 64.074,Z 493.572,A -85,B 0,C 180,E1 -28403.092,E2 -28403.092} C_VEL
LIN {X 0,Y 63.416,Z 501.732,A -85,B 0,C 180,E1 -28412.415,E2 -28412.415} C_VEL
LIN {X 0,Y 64.419,Z 509.84,A -85,B 0,C 180,E1 -28424.137,E2 -28424.137} C_VEL
LIN {X 0,Y 67.356,Z 515.646,A -85,B 0,C 180,E1 -28434.014,E2 -28434.014} C_VEL
LIN {X 0,Y 72.119,Z 520.231,A -85,B 0,C 180,E1 -28442.796,E2 -28442.796} C_VEL
LIN {X 0,Y 78.627,Z 523.85,A -85,B 0,C 180,E1 -28450.586,E2 -28450.586} C_VEL
LIN {X 0,Y 83.263,Z 525.564,A -85,B 0,C 180,E1 -28454.671,E2 -28454.671} C_VEL
LIN {X 0,Y 89.017,Z 527.006,A -85,B 0,C 180,E1 -28458.703,E2 -28458.703} C_VEL
LIN {X 0,Y 100.689,Z 528.459,A -85,B 0,C 180,E1 -28464.761,E2 -28464.761} C_VEL
LIN {X 0,Y 110.999,Z 528.473,A -85,B 0,C 180,E1 -28468.652,E2 -28468.652} C_VEL
LIN {X 0,Y 109.837,Z 528.694,A -85,B 0,C 180,E1 -28469.755,E2 -28469.755} C_VEL
LIN {X 0,Y 100.671,Z 529.428,A -85,B 0,C 180,E1 -28473.118,E2 -28473.118} C_VEL
LIN {X 0,Y 89.856,Z 529.256,A -85,B 0,C 180,E1 -28478.562,E2 -28478.562} C_VEL
LIN {X 0,Y 80.406,Z 527.891,A -85,B 0,C 180,E1 -28485.65,E2 -28485.65} C_VEL
LIN {X 0,Y 72.659,Z 525.3,A -85,B 0,C 180,E1 -28494.54,E2 -28494.54} C_VEL
LIN {X 0,Y 67.541,Z 521.414,A -85,B 0,C 180,E1 -28505.417,E2 -28505.417} C_VEL
LIN {X 0,Y 65.517,Z 516.136,A -85,B 0,C 180,E1 -28517.623,E2 -28517.623} C_VEL
LIN {X 0,Y 65.637,Z 512.793,A -85,B 0,C 180,E1 -28523.864,E2 -28523.864} C_VEL
LIN {X 0,Y 65.396,Z 508.582,A -85,B 0,C 180,E1 -28530.01,E2 -28530.01} C_VEL
LIN {X 0,Y 65.2,Z 502.011,A -85,B 0,C 180,E1 -28537.753,E2 -28537.753} C_VEL
LIN {X 0,Y 66.194,Z 492.791,A -85,B 0,C 180,E1 -28546.548,E2 -28546.548} C_VEL
LIN {X 0,Y 68.252,Z 482.13,A -85,B 0,C 180,E1 -28554.331,E2 -28554.331} C_VEL
LIN {X 0,Y 70.589,Z 472.206,A -85,B 0,C 180,E1 -28559.863,E2 -28559.863} C_VEL
LIN {X 0,Y 73.155,Z 461.546,A -85,B 0,C 180,E1 -28564.368,E2 -28564.368} C_VEL
LIN {X 0,Y 75.892,Z 448.873,A -85,B 0,C 180,E1 -28568.271,E2 -28568.271} C_VEL
LIN {X 0,Y 78.306,Z 435.023,A -85,B 0,C 180,E1 -28571.238,E2 -28571.238} C_VEL
LIN {X 0,Y 80.498,Z 415.202,A -85,B 0,C 180,E1 -28573.873,E2 -28573.873} C_VEL
LIN {X 0,Y 82.592,Z 393.618,A -85,B 0,C 180,E1 -28576.396,E2 -28576.396} C_VEL
LIN {X 0,Y 81.929,Z 376.468,A -85,B 0,C 180,E1 -28579.071,E2 -28579.071} C_VEL
LIN {X 0,Y 76.691,Z 356.623,A -85,B 0,C 180,E1 -28584.114,E2 -28584.114} C_VEL
LIN {X 0,Y 72.725,Z 347.247,A -85,B 0,C 180,E1 -28587.473,E2 -28587.473} C_VEL
LIN {X 0,Y 68.499,Z 338.978,A -85,B 0,C 180,E1 -28591.298,E2 -28591.298} C_VEL
LIN {X 0,Y 66.84,Z 336.033,A -85,B 0,C 180,E1 -28592.917,E2 -28592.917} C_VEL
LIN {X 0,Y 65.435,Z 333.326,A -85,B 0,C 180,E1 -28594.413,E2 -28594.413} C_VEL
LIN {X 0,Y 65.253,Z 332.353,A -85,B 0,C 180,E1 -28594.904,E2 -28594.904} C_VEL
LIN {X 0,Y 65.584,Z 332.308,A -85,B 0,C 180,E1 -28604.692,E2 -28604.692} C_VEL
LIN {X 0,Y 65.878,Z 332.27,A -85,B 0,C 180,E1 -28613.873,E2 -28613.873} C_VEL
LIN {X 0,Y 66.447,Z 332.205,A -85,B 0,C 180,E1 -28619.997,E2 -28619.997} C_VEL
LIN {X 0,Y 65.69,Z 332.297,A -85,B 0,C 180,E1 -28632.352,E2 -28632.352} C_VEL
LIN {X 0,Y 65.338,Z 332.337,A -85,B 0,C 180,E1 -28638.823,E2 -28638.823} C_VEL
LIN {X 0,Y 65.202,Z 332.356,A -85,B 0,C 180,E1 -28645.203,E2 -28645.203} C_VEL
LIN {X 0,Y 64.979,Z 332.405,A -85,B 0,C 180,E1 -28648.642,E2 -28648.642} C_VEL
LIN {X 0,Y 64.197,Z 332.513,A -85,B 0,C 180,E1 -28652.056,E2 -28652.056} C_VEL
LIN {X 0,Y 62.415,Z 332.735,A -85,B 0,C 180,E1 -28657.214,E2 -28657.214} C_VEL
LIN {X 0,Y 58.326,Z 333.217,A -85,B 0,C 180,E1 -28670.393,E2 -28670.393} C_VEL
LIN {X 0,Y 58.032,Z 333.244,A -85,B 0,C 180,E1 -28674.464,E2 -28674.464} C_VEL
LIN {X 0,Y 58.151,Z 333.232,A -85,B 0,C 180,E1 -28681.081,E2 -28681.081} C_VEL
LIN {X 0,Y 58.516,Z 333.196,A -85,B 0,C 180,E1 -28693.9,E2 -28693.9} C_VEL
LIN {X 0,Y 58.655,Z 333.173,A -85,B 0,C 180,E1 -28696.125,E2 -28696.125} C_VEL
LIN {X 0,Y 58.862,Z 333.15,A -85,B 0,C 180,E1 -28703.778,E2 -28703.778} C_VEL
LIN {X 0,Y 60.006,Z 336.012,A -85,B 0,C 180,E1 -28705.479,E2 -28705.479} C_VEL
LIN {X 0,Y 61.965,Z 338.158,A -85,B 0,C 180,E1 -28707.524,E2 -28707.524} C_VEL
LIN {X 0,Y 67.651,Z 350.553,A -85,B 0,C 180,E1 -28713.806,E2 -28713.806} C_VEL
LIN {X 0,Y 72.478,Z 363.546,A -85,B 0,C 180,E1 -28718.65,E2 -28718.65} C_VEL
LIN {X 0,Y 77.142,Z 377.375,A -85,B 0,C 180,E1 -28722.777,E2 -28722.777} C_VEL
LIN {X 0,Y 71.936,Z 423.379,A -85,B 0,C 180,E1 -28728.571,E2 -28728.571} C_VEL
LIN {X 0,Y 69.434,Z 437.925,A -85,B 0,C 180,E1 -28731.582,E2 -28731.582} C_VEL
LIN {X 0,Y 66.625,Z 450.6,A -85,B 0,C 180,E1 -28735.488,E2 -28735.488} C_VEL
LIN {X 0,Y 63.606,Z 462.744,A -85,B 0,C 180,E1 -28740.694,E2 -28740.694} C_VEL
LIN {X 0,Y 60.777,Z 474.104,A -85,B 0,C 180,E1 -28747.351,E2 -28747.351} C_VEL
LIN {X 0,Y 58.324,Z 484.784,A -85,B 0,C 180,E1 -28755.731,E2 -28755.731} C_VEL
LIN {X 0,Y 57.005,Z 493.053,A -85,B 0,C 180,E1 -28764.158,E2 -28764.158} C_VEL
LIN {X 0,Y 56.523,Z 501.028,A -85,B 0,C 180,E1 -28774.282,E2 -28774.282} C_VEL
LIN {X 0,Y 57.825,Z 508.853,A -85,B 0,C 180,E1 -28786.413,E2 -28786.413} C_VEL
LIN {X 0,Y 61.023,Z 514.608,A -85,B 0,C 180,E1 -28796.702,E2 -28796.702} C_VEL
LIN {X 0,Y 66.282,Z 519.463,A -85,B 0,C 180,E1 -28806.09,E2 -28806.09} C_VEL
LIN {X 0,Y 72.091,Z 522.82,A -85,B 0,C 180,E1 -28812.934,E2 -28812.934} C_VEL
LIN {X 0,Y 81.174,Z 526.121,A -85,B 0,C 180,E1 -28820.265,E2 -28820.265} C_VEL
LIN {X 0,Y 87.149,Z 527.478,A -85,B 0,C 180,E1 -28823.782,E2 -28823.782} C_VEL
LIN {X 0,Y 97.899,Z 528.856,A -85,B 0,C 180,E1 -28828.624,E2 -28828.624} C_VEL
LIN {X 0,Y 96.984,Z 528.946,A -85,B 0,C 180,E1 -28829.613,E2 -28829.613} C_VEL
LIN {X 0,Y 85.638,Z 528.433,A -85,B 0,C 180,E1 -28834.871,E2 -28834.871} C_VEL
LIN {X 0,Y 75.543,Z 526.756,A -85,B 0,C 180,E1 -28841.923,E2 -28841.923} C_VEL
LIN {X 0,Y 67.112,Z 523.79,A -85,B 0,C 180,E1 -28851.091,E2 -28851.091} C_VEL
LIN {X 0,Y 61.355,Z 519.594,A -85,B 0,C 180,E1 -28862.745,E2 -28862.745} C_VEL
LIN {X 0,Y 58.942,Z 513.951,A -85,B 0,C 180,E1 -28876.216,E2 -28876.216} C_VEL
LIN {X 0,Y 58.931,Z 510.488,A -85,B 0,C 180,E1 -28883.162,E2 -28883.162} C_VEL
LIN {X 0,Y 58.562,Z 505.982,A -85,B 0,C 180,E1 -28890.011,E2 -28890.011} C_VEL
LIN {X 0,Y 58.451,Z 497.412,A -85,B 0,C 180,E1 -28900.401,E2 -28900.401} C_VEL
LIN {X 0,Y 59.717,Z 488.667,A -85,B 0,C 180,E1 -28908.857,E2 -28908.857} C_VEL
LIN {X 0,Y 62.065,Z 477.7,A -85,B 0,C 180,E1 -28916.941,E2 -28916.941} C_VEL
LIN {X 0,Y 64.742,Z 466.944,A -85,B 0,C 180,E1 -28922.881,E2 -28922.881} C_VEL
LIN {X 0,Y 67.59,Z 455.113,A -85,B 0,C 180,E1 -28927.661,E2 -28927.661} C_VEL
LIN {X 0,Y 70.349,Z 441.824,A -85,B 0,C 180,E1 -28931.448,E2 -28931.448} C_VEL
LIN {X 0,Y 72.247,Z 429.351,A -85,B 0,C 180,E1 -28933.883,E2 -28933.883} C_VEL
LIN {X 0,Y 76.084,Z 394.609,A -85,B 0,C 180,E1 -28938.304,E2 -28938.304} C_VEL
LIN {X 0,Y 75.567,Z 378.094,A -85,B 0,C 180,E1 -28941.11,E2 -28941.11} C_VEL
LIN {X 0,Y 70.753,Z 359.295,A -85,B 0,C 180,E1 -28946.298,E2 -28946.298} C_VEL
LIN {X 0,Y 66.418,Z 349.006,A -85,B 0,C 180,E1 -28950.603,E2 -28950.603} C_VEL
LIN {X 0,Y 62.32,Z 340.973,A -85,B 0,C 180,E1 -28955.036,E2 -28955.036} C_VEL
LIN {X 0,Y 60.057,Z 337.088,A -85,B 0,C 180,E1 -28957.644,E2 -28957.644} C_VEL
LIN {X 0,Y 58.567,Z 334.53,A -85,B 0,C 180,E1 -28959.533,E2 -28959.533} C_VEL
LIN {X 0,Y 58.279,Z 333.225,A -85,B 0,C 180,E1 -28960.275,E2 -28960.275} C_VEL
LIN {X 0,Y 58.565,Z 333.181,A -85,B 0,C 180,E1 -28966.11,E2 -28966.11} C_VEL
LIN {X 0,Y 58.76,Z 333.157,A -85,B 0,C 180,E1 -28973.127,E2 -28973.127} C_VEL
LIN {X 0,Y 59.338,Z 333.09,A -85,B 0,C 180,E1 -28979.997,E2 -28979.997} C_VEL
LIN {X 0,Y 58.76,Z 333.166,A -85,B 0,C 180,E1 -28986.866,E2 -28986.866} C_VEL
LIN {X 0,Y 58.458,Z 333.202,A -85,B 0,C 180,E1 -28995.87,E2 -28995.87} C_VEL
LIN {X 0,Y 58.012,Z 333.237,A -85,B 0,C 180,E1 -29005.189,E2 -29005.189} C_VEL
LIN {X 0,Y 58.135,Z 333.243,A -85,B 0,C 180,E1 -29012.184,E2 -29012.184} C_VEL
LIN {X 0,Y 58.027,Z 333.25,A -85,B 0,C 180,E1 -29017.266,E2 -29017.266} C_VEL
LIN {X 0,Y 58.024,Z 333.254,A -85,B 0,C 180,E1 -29026.608,E2 -29026.608} C_VEL
LIN {X 0,Y 58.032,Z 333.244,A -85,B 0,C 180,E1 -29034.464,E2 -29034.464} C_VEL
LIN {X 0,Y 57.381,Z 333.336,A -85,B 0,C 180,E1 -29038.283,E2 -29038.283} C_VEL
LIN {X 0,Y 55.846,Z 333.527,A -85,B 0,C 180,E1 -29042.002,E2 -29042.002} C_VEL
LIN {X 0,Y 51.954,Z 334.014,A -85,B 0,C 180,E1 -29051.319,E2 -29051.319} C_VEL
LIN {X 0,Y 51.574,Z 334.055,A -85,B 0,C 180,E1 -29055.827,E2 -29055.827} C_VEL
LIN {X 0,Y 51.606,Z 334.05,A -85,B 0,C 180,E1 -29056.201,E2 -29056.201} C_VEL
LIN {X 0,Y 52.495,Z 336.741,A -85,B 0,C 180,E1 -29058.159,E2 -29058.159} C_VEL
LIN {X 0,Y 54.838,Z 339.34,A -85,B 0,C 180,E1 -29061.525,E2 -29061.525} C_VEL
LIN {X 0,Y 56.949,Z 342.58,A -85,B 0,C 180,E1 -29064.451,E2 -29064.451} C_VEL
LIN {X 0,Y 58.265,Z 344.915,A -85,B 0,C 180,E1 -29066.185,E2 -29066.185} C_VEL
LIN {X 0,Y 62.367,Z 354.436,A -85,B 0,C 180,E1 -29071.377,E2 -29071.377} C_VEL
LIN {X 0,Y 67.018,Z 367.482,A -85,B 0,C 180,E1 -29076.71,E2 -29076.71} C_VEL
LIN {X 0,Y 70.661,Z 379.241,A -85,B 0,C 180,E1 -29080.567,E2 -29080.567} C_VEL
LIN {X 0,Y 65.169,Z 424.107,A -85,B 0,C 180,E1 -29086.589,E2 -29086.589} C_VEL
LIN {X 0,Y 62.682,Z 437.805,A -85,B 0,C 180,E1 -29089.643,E2 -29089.643} C_VEL
LIN {X 0,Y 59.613,Z 450.884,A -85,B 0,C 180,E1 -29093.989,E2 -29093.989} C_VEL
LIN {X 0,Y 56.572,Z 462.691,A -85,B 0,C 180,E1 -29099.593,E2 -29099.593} C_VEL
LIN {X 0,Y 53.703,Z 473.606,A -85,B 0,C 180,E1 -29106.727,E2 -29106.727} C_VEL
LIN {X 0,Y 51.431,Z 483.188,A -85,B 0,C 180,E1 -29115.08,E2 -29115.08} C_VEL
LIN {X 0,Y 49.966,Z 492.627,A -85,B 0,C 180,E1 -29125.768,E2 -29125.768} C_VEL
LIN {X 0,Y 49.747,Z 500.597,A -85,B 0,C 180,E1 -29137.143,E2 -29137.143} C_VEL
LIN {X 0,Y 51.357,Z 507.642,A -85,B 0,C 180,E1 -29149.166,E2 -29149.166} C_VEL
LIN {X 0,Y 56.279,Z 514.926,A -85,B 0,C 180,E1 -29162.903,E2 -29162.903} C_VEL
LIN {X 0,Y 63.057,Z 520.07,A -85,B 0,C 180,E1 -29172.883,E2 -29172.883} C_VEL
LIN {X 0,Y 73.822,Z 524.856,A -85,B 0,C 180,E1 -29182.387,E2 -29182.387} C_VEL
LIN {X 0,Y 84.606,Z 527.696,A -85,B 0,C 180,E1 -29188.39,E2 -29188.39} C_VEL
LIN {X 0,Y 81.818,Z 527.462,A -85,B 0,C 180,E1 -29190.823,E2 -29190.823} C_VEL
LIN {X 0,Y 71.058,Z 525.434,A -85,B 0,C 180,E1 -29197.721,E2 -29197.721} C_VEL
LIN {X 0,Y 61.887,Z 522.182,A -85,B 0,C 180,E1 -29207.068,E2 -29207.068} C_VEL
LIN {X 0,Y 55.37,Z 517.648,A -85,B 0,C 180,E1 -29219.505,E2 -29219.505} C_VEL
LIN {X 0,Y 52.749,Z 513.126,A -85,B 0,C 180,E1 -29231.084,E2 -29231.084} C_VEL
LIN {X 0,Y 52.303,Z 507.945,A -85,B 0,C 180,E1 -29242.291,E2 -29242.291} C_VEL
LIN {X 0,Y 51.886,Z 504.445,A -85,B 0,C 180,E1 -29248.072,E2 -29248.072} C_VEL
LIN {X 0,Y 51.528,Z 497.337,A -85,B 0,C 180,E1 -29257.851,E2 -29257.851} C_VEL
LIN {X 0,Y 52.5,Z 488.767,A -85,B 0,C 180,E1 -29267.5,E2 -29267.5} C_VEL
LIN {X 0,Y 54.642,Z 478.437,A -85,B 0,C 180,E1 -29276.353,E2 -29276.353} C_VEL
LIN {X 0,Y 57.501,Z 467.38,A -85,B 0,C 180,E1 -29283.377,E2 -29283.377} C_VEL
LIN {X 0,Y 60.399,Z 455.811,A -85,B 0,C 180,E1 -29288.723,E2 -29288.723} C_VEL
LIN {X 0,Y 63.315,Z 442.938,A -85,B 0,C 180,E1 -29292.842,E2 -29292.842} C_VEL
LIN {X 0,Y 65.406,Z 430.21,A -85,B 0,C 180,E1 -29295.67,E2 -29295.67} C_VEL
LIN {X 0,Y 69.579,Z 394.64,A -85,B 0,C 180,E1 -29300.595,E2 -29300.595} C_VEL
LIN {X 0,Y 69.207,Z 379.786,A -85,B 0,C 180,E1 -29303.362,E2 -29303.362} C_VEL
LIN {X 0,Y 64.849,Z 361.748,A -85,B 0,C 180,E1 -29308.978,E2 -29308.978} C_VEL
LIN {X 0,Y 60.221,Z 350.656,A -85,B 0,C 180,E1 -29314.379,E2 -29314.379} C_VEL
LIN {X 0,Y 55.878,Z 342.332,A -85,B 0,C 180,E1 -29320.001,E2 -29320.001} C_VEL
LIN {X 0,Y 53.514,Z 338.338,A -85,B 0,C 180,E1 -29323.546,E2 -29323.546} C_VEL
LIN {X 0,Y 51.906,Z 335.613,A -85,B 0,C 180,E1 -29326.29,E2 -29326.29} C_VEL
LIN {X 0,Y 51.5,Z 334.065,A -85,B 0,C 180,E1 -29327.685,E2 -29327.685} C_VEL
LIN {X 0,Y 52.222,Z 333.976,A -85,B 0,C 180,E1 -29339.996,E2 -29339.996} C_VEL
LIN {X 0,Y 51.634,Z 334.052,A -85,B 0,C 180,E1 -29347.819,E2 -29347.819} C_VEL
LIN {X 0,Y 51.341,Z 334.086,A -85,B 0,C 180,E1 -29356.596,E2 -29356.596} C_VEL
LIN {X 0,Y 51,Z 334.131,A -85,B 0,C 180,E1 -29364.415,E2 -29364.415} C_VEL
LIN {X 0,Y 51.014,Z 334.124,A -85,B 0,C 180,E1 -29374.235,E2 -29374.235} C_VEL
LIN {X 0,Y 50.989,Z 334.125,A -85,B 0,C 180,E1 -29383.559,E2 -29383.559} C_VEL
LIN {X 0,Y 51.034,Z 334.127,A -85,B 0,C 180,E1 -29395.71,E2 -29395.71} C_VEL
LIN {X 0,Y 51.024,Z 334.129,A -85,B 0,C 180,E1 -29405.582,E2 -29405.582} C_VEL
LIN {X 0,Y 51.574,Z 334.055,A -85,B 0,C 180,E1 -29415.827,E2 -29415.827} C_VEL
LIN {X 0,Y 52.949,Z 334.681,A -85,B 0,C 180,E1 -29418.071,E2 -29418.071} C_VEL
LIN {X 0,Y 54.696,Z 336.798,A -85,B 0,C 180,E1 -29420.655,E2 -29420.655} C_VEL
LIN {X 0,Y 56.202,Z 340.71,A -85,B 0,C 180,E1 -29423.264,E2 -29423.264} C_VEL
LIN {X 0,Y 57.256,Z 346.528,A -85,B 0,C 180,E1 -29425.453,E2 -29425.453} C_VEL
LIN {X 0,Y 58.015,Z 359.799,A -85,B 0,C 180,E1 -29429.521,E2 -29429.521} C_VEL
LIN {X 0,Y 58.398,Z 361.927,A -85,B 0,C 180,E1 -29430.333,E2 -29430.333} C_VEL
LIN {X 0,Y 62.677,Z 374.971,A -85,B 0,C 180,E1 -29435.821,E2 -29435.821} C_VEL
LIN {X 0,Y 64.33,Z 380.215,A -85,B 0,C 180,E1 -29437.754,E2 -29437.754} C_VEL
LIN {X 0,Y 58.531,Z 424.531,A -85,B 0,C 180,E1 -29444.141,E2 -29444.141} C_VEL
LIN {X 0,Y 56.089,Z 437.169,A -85,B 0,C 180,E1 -29447.184,E2 -29447.184} C_VEL
LIN {X 0,Y 52.948,Z 449.924,A -85,B 0,C 180,E1 -29451.709,E2 -29451.709} C_VEL
LIN {X 0,Y 49.551,Z 462.386,A -85,B 0,C 180,E1 -29458.236,E2 -29458.236} C_VEL
LIN {X 0,Y 46.682,Z 472.833,A -85,B 0,C 180,E1 -29465.868,E2 -29465.868} C_VEL
LIN {X 0,Y 44.219,Z 483.038,A -85,B 0,C 180,E1 -29475.951,E2 -29475.951} C_VEL
LIN {X 0,Y 42.972,Z 491.931,A -85,B 0,C 180,E1 -29487.51,E2 -29487.51} C_VEL
LIN {X 0,Y 42.965,Z 498.657,A -85,B 0,C 180,E1 -29498.41,E2 -29498.41} C_VEL
LIN {X 0,Y 45.192,Z 506.624,A -85,B 0,C 180,E1 -29513.307,E2 -29513.307} C_VEL
LIN {X 0,Y 50.96,Z 514.047,A -85,B 0,C 180,E1 -29527.931,E2 -29527.931} C_VEL
LIN {X 0,Y 59.445,Z 519.884,A -85,B 0,C 180,E1 -29538.999,E2 -29538.999} C_VEL
LIN {X 0,Y 66.627,Z 523.183,A -85,B 0,C 180,E1 -29544.96,E2 -29544.96} C_VEL
LIN {X 0,Y 72.867,Z 525.376,A -85,B 0,C 180,E1 -29548.836,E2 -29548.836} C_VEL
LIN {X 0,Y 72.593,Z 525.353,A -85,B 0,C 180,E1 -29549.415,E2 -29549.415} C_VEL
LIN {X 0,Y 61.808,Z 522.362,A -85,B 0,C 180,E1 -29557.28,E2 -29557.28} C_VEL
LIN {X 0,Y 52.912,Z 518.133,A -85,B 0,C 180,E1 -29568.407,E2 -29568.407} C_VEL
LIN {X 0,Y 47.375,Z 512.617,A -85,B 0,C 180,E1 -29583.592,E2 -29583.592} C_VEL
LIN {X 0,Y 45.735,Z 506.375,A -85,B 0,C 180,E1 -29598.941,E2 -29598.941} C_VEL
LIN {X 0,Y 45.322,Z 502.865,A -85,B 0,C 180,E1 -29605.568,E2 -29605.568} C_VEL
LIN {X 0,Y 44.72,Z 495.553,A -85,B 0,C 180,E1 -29616.783,E2 -29616.783} C_VEL
LIN {X 0,Y 45.898,Z 485.328,A -85,B 0,C 180,E1 -29629.373,E2 -29629.373} C_VEL
LIN {X 0,Y 48.518,Z 474.058,A -85,B 0,C 180,E1 -29639.636,E2 -29639.636} C_VEL
LIN {X 0,Y 51.912,Z 461.627,A -85,B 0,C 180,E1 -29647.544,E2 -29647.544} C_VEL
LIN {X 0,Y 55.012,Z 449.656,A -85,B 0,C 180,E1 -29652.753,E2 -29652.753} C_VEL
LIN {X 0,Y 57.872,Z 435.914,A -85,B 0,C 180,E1 -29656.783,E2 -29656.783} C_VEL
LIN {X 0,Y 59.909,Z 422.067,A -85,B 0,C 180,E1 -29659.373,E2 -29659.373} C_VEL
LIN {X 0,Y 63.227,Z 394.316,A -85,B 0,C 180,E1 -29663.385,E2 -29663.385} C_VEL
LIN {X 0,Y 63.004,Z 381.243,A -85,B 0,C 180,E1 -29666.097,E2 -29666.097} C_VEL
LIN {X 0,Y 59.065,Z 364.3,A -85,B 0,C 180,E1 -29672.099,E2 -29672.099} C_VEL
LIN {X 0,Y 55.115,Z 354.513,A -85,B 0,C 180,E1 -29677.505,E2 -29677.505} C_VEL
LIN {X 0,Y 51.489,Z 347.107,A -85,B 0,C 180,E1 -29683.237,E2 -29683.237} C_VEL
LIN {X 0,Y 49.062,Z 342.812,A -85,B 0,C 180,E1 -29687.669,E2 -29687.669} C_VEL
LIN {X 0,Y 47.756,Z 340.037,A -85,B 0,C 180,E1 -29690.487,E2 -29690.487} C_VEL
LIN {X 0,Y 45.607,Z 337.622,A -85,B 0,C 180,E1 -29695.023,E2 -29695.023} C_VEL
LIN {X 0,Y 44.871,Z 334.896,A -85,B 0,C 180,E1 -29697.751,E2 -29697.751} C_VEL
LIN {X 0,Y 45.096,Z 334.862,A -85,B 0,C 180,E1 -29699.996,E2 -29699.996} C_VEL
LIN {X 0,Y 44.48,Z 334.937,A -85,B 0,C 180,E1 -29709.086,E2 -29709.086} C_VEL
LIN {X 0,Y 44.109,Z 334.981,A -85,B 0,C 180,E1 -29718.577,E2 -29718.577} C_VEL
LIN {X 0,Y 43.816,Z 335.019,A -85,B 0,C 180,E1 -29728.758,E2 -29728.758} C_VEL
LIN {X 0,Y 43.801,Z 335.029,A -85,B 0,C 180,E1 -29739.921,E2 -29739.921} C_VEL
LIN {X 0,Y 43.847,Z 335.014,A -85,B 0,C 180,E1 -29753.258,E2 -29753.258} C_VEL
LIN {X 0,Y 43.903,Z 335.101,A -85,B 0,C 180,E1 -29763.613,E2 -29763.613} C_VEL
LIN {X 0,Y 44.922,Z 337.738,A -85,B 0,C 180,E1 -29767.101,E2 -29767.101} C_VEL
LIN {X 0,Y 47.189,Z 339.897,A -85,B 0,C 180,E1 -29772.043,E2 -29772.043} C_VEL
LIN {X 0,Y 48.017,Z 340.693,A -85,B 0,C 180,E1 -29773.609,E2 -29773.609} C_VEL
LIN {X 0,Y 49.997,Z 343.858,A -85,B 0,C 180,E1 -29777.371,E2 -29777.371} C_VEL
LIN {X 0,Y 51.234,Z 345.433,A -85,B 0,C 180,E1 -29779.331,E2 -29779.331} C_VEL
LIN {X 0,Y 53.402,Z 348.875,A -85,B 0,C 180,E1 -29782.718,E2 -29782.718} C_VEL
LIN {X 0,Y 57.069,Z 358.034,A -85,B 0,C 180,E1 -29788.412,E2 -29788.412} C_VEL
LIN {X 0,Y 58.398,Z 361.927,A -85,B 0,C 180,E1 -29790.333,E2 -29790.333} C_VEL
LIN {X 0,Y 59.19,Z 367.527,A -85,B 0,C 180,E1 -29792.15,E2 -29792.15} C_VEL
LIN {X 0,Y 59.21,Z 373.351,A -85,B 0,C 180,E1 -29793.452,E2 -29793.452} C_VEL
LIN {X 0,Y 57.76,Z 385.242,A -85,B 0,C 180,E1 -29795.191,E2 -29795.191} C_VEL
LIN {X 0,Y 56.446,Z 393.203,A -85,B 0,C 180,E1 -29796.191,E2 -29796.191} C_VEL
LIN {X 0,Y 51.947,Z 424.994,A -85,B 0,C 180,E1 -29801.248,E2 -29801.248} C_VEL
LIN {X 0,Y 49.033,Z 438.967,A -85,B 0,C 180,E1 -29804.974,E2 -29804.974} C_VEL
LIN {X 0,Y 45.52,Z 451.985,A -85,B 0,C 180,E1 -29810.37,E2 -29810.37} C_VEL
LIN {X 0,Y 41.838,Z 464.459,A -85,B 0,C 180,E1 -29818.139,E2 -29818.139} C_VEL
LIN {X 0,Y 38.857,Z 475.012,A -85,B 0,C 180,E1 -29827.701,E2 -29827.701} C_VEL
LIN {X 0,Y 36.526,Z 485.912,A -85,B 0,C 180,E1 -29841.761,E2 -29841.761} C_VEL
LIN {X 0,Y 36.078,Z 493.274,A -85,B 0,C 180,E1 -29854.011,E2 -29854.011} C_VEL
LIN {X 0,Y 37.736,Z 502.302,A -85,B 0,C 180,E1 -29871.976,E2 -29871.976} C_VEL
LIN {X 0,Y 42.495,Z 509.635,A -85,B 0,C 180,E1 -29887.28,E2 -29887.28} C_VEL
LIN {X 0,Y 50.827,Z 516.378,A -85,B 0,C 180,E1 -29900.232,E2 -29900.232} C_VEL
LIN {X 0,Y 60.625,Z 521.513,A -85,B 0,C 180,E1 -29908.801,E2 -29908.801} C_VEL
LIN {X 0,Y 59.23,Z 521.129,A -85,B 0,C 180,E1 -29910.768,E2 -29910.768} C_VEL
LIN {X 0,Y 48.052,Z 516.059,A -85,B 0,C 180,E1 -29923.031,E2 -29923.031} C_VEL
LIN {X 0,Y 41.499,Z 510.171,A -85,B 0,C 180,E1 -29939.487,E2 -29939.487} C_VEL
LIN {X 0,Y 39.454,Z 504.636,A -85,B 0,C 180,E1 -29954.521,E2 -29954.521} C_VEL
LIN {X 0,Y 39.151,Z 502.462,A -85,B 0,C 180,E1 -29959.677,E2 -29959.677} C_VEL
LIN {X 0,Y 38.105,Z 496.881,A -85,B 0,C 180,E1 -29970.017,E2 -29970.017} C_VEL
LIN {X 0,Y 38.225,Z 488.413,A -85,B 0,C 180,E1 -29983.302,E2 -29983.302} C_VEL
LIN {X 0,Y 39.951,Z 479.11,A -85,B 0,C 180,E1 -29994.795,E2 -29994.795} C_VEL
LIN {X 0,Y 43.047,Z 467.781,A -85,B 0,C 180,E1 -30004.869,E2 -30004.869} C_VEL
LIN {X 0,Y 46.194,Z 456.677,A -85,B 0,C 180,E1 -30011.743,E2 -30011.743} C_VEL
LIN {X 0,Y 49.384,Z 444.649,A -85,B 0,C 180,E1 -30016.845,E2 -30016.845} C_VEL
LIN {X 0,Y 52.059,Z 431.431,A -85,B 0,C 180,E1 -30020.55,E2 -30020.55} C_VEL
LIN {X 0,Y 56.422,Z 400.095,A -85,B 0,C 180,E1 -30025.726,E2 -30025.726} C_VEL
LIN {X 0,Y 56.996,Z 393.726,A -85,B 0,C 180,E1 -30026.821,E2 -30026.821} C_VEL
LIN {X 0,Y 56.89,Z 382.737,A -85,B 0,C 180,E1 -30029.358,E2 -30029.358} C_VEL
LIN {X 0,Y 53.606,Z 367.48,A -85,B 0,C 180,E1 -30035.434,E2 -30035.434} C_VEL
LIN {X 0,Y 50.15,Z 358.217,A -85,B 0,C 180,E1 -30041.362,E2 -30041.362} C_VEL
LIN {X 0,Y 46.97,Z 351.313,A -85,B 0,C 180,E1 -30047.575,E2 -30047.575} C_VEL
LIN {X 0,Y 44.012,Z 345.498,A -85,B 0,C 180,E1 -30054.612,E2 -30054.612} C_VEL
LIN {X 0,Y 42.161,Z 342.553,A -85,B 0,C 180,E1 -30059.995,E2 -30059.995} C_VEL
LIN {X 0,Y 41.735,Z 341.236,A -85,B 0,C 180,E1 -30061.805,E2 -30061.805} C_VEL
LIN {X 0,Y 37.849,Z 338.528,A -85,B 0,C 180,E1 -30079.57,E2 -30079.57} C_VEL
LIN {X 0,Y 37.286,Z 337.806,A -85,B 0,C 180,E1 -30088.107,E2 -30088.107} C_VEL
LIN {X 0,Y 37.493,Z 338.298,A -85,B 0,C 180,E1 -30099.947,E2 -30099.947} C_VEL
LIN {X 0,Y 41.233,Z 341.827,A -85,B 0,C 180,E1 -30120.479,E2 -30120.479} C_VEL
LIN {X 0,Y 42.944,Z 344.951,A -85,B 0,C 180,E1 -30126.358,E2 -30126.358} C_VEL
LIN {X 0,Y 44.706,Z 346.698,A -85,B 0,C 180,E1 -30130.587,E2 -30130.587} C_VEL
LIN {X 0,Y 47.7,Z 351.461,A -85,B 0,C 180,E1 -30136.949,E2 -30136.949} C_VEL
LIN {X 0,Y 49.081,Z 353.883,A -85,B 0,C 180,E1 -30139.467,E2 -30139.467} C_VEL
LIN {X 0,Y 52.073,Z 361.966,A -85,B 0,C 180,E1 -30145.073,E2 -30145.073} C_VEL
LIN {X 0,Y 56.254,Z 375.505,A -85,B 0,C 180,E1 -30151.982,E2 -30151.982} C_VEL
LIN {X 0,Y 57.987,Z 381.963,A -85,B 0,C 180,E1 -30154.597,E2 -30154.597} C_VEL
LIN {X 0,Y 56.446,Z 393.203,A -85,B 0,C 180,E1 -30156.191,E2 -30156.191} C_VEL
LIN {X 0,Y 55.06,Z 398.92,A -85,B 0,C 180,E1 -30156.659,E2 -30156.659} C_VEL
LIN {X 0,Y 48.256,Z 415.404,A -85,B 0,C 180,E1 -30156.376,E2 -30156.376} C_VEL
LIN {X 0,Y 46.437,Z 421.032,A -85,B 0,C 180,E1 -30156.709,E2 -30156.709} C_VEL
LIN {X 0,Y 46.018,Z 422.947,A -85,B 0,C 180,E1 -30157.002,E2 -30157.002} C_VEL
LIN {X 0,Y 43.318,Z 435.725,A -85,B 0,C 180,E1 -30160.292,E2 -30160.292} C_VEL
LIN {X 0,Y 39.672,Z 448.78,A -85,B 0,C 180,E1 -30165.599,E2 -30165.599} C_VEL
LIN {X 0,Y 36.115,Z 460.269,A -85,B 0,C 180,E1 -30172.883,E2 -30172.883} C_VEL
LIN {X 0,Y 32.226,Z 472.73,A -85,B 0,C 180,E1 -30185.14,E2 -30185.14} C_VEL
LIN {X 0,Y 29.862,Z 482.718,A -85,B 0,C 180,E1 -30199.678,E2 -30199.678} C_VEL
LIN {X 0,Y 29.412,Z 492.201,A -85,B 0,C 180,E1 -30218.116,E2 -30218.116} C_VEL
LIN {X 0,Y 31.576,Z 500.3,A -85,B 0,C 180,E1 -30236.817,E2 -30236.817} C_VEL
LIN {X 0,Y 37.244,Z 507.863,A -85,B 0,C 180,E1 -30253.649,E2 -30253.649} C_VEL
LIN {X 0,Y 46.701,Z 515.088,A -85,B 0,C 180,E1 -30266.843,E2 -30266.843} C_VEL
LIN {X 0,Y 47.636,Z 515.658,A -85,B 0,C 180,E1 -30267.763,E2 -30267.763} C_VEL
LIN {X 0,Y 48.907,Z 516.486,A -85,B 0,C 180,E1 -30270.471,E2 -30270.471} C_VEL
LIN {X 0,Y 39.318,Z 510.899,A -85,B 0,C 180,E1 -30284.387,E2 -30284.387} C_VEL
LIN {X 0,Y 34.704,Z 505.815,A -85,B 0,C 180,E1 -30299.608,E2 -30299.608} C_VEL
LIN {X 0,Y 32.998,Z 500.61,A -85,B 0,C 180,E1 -30314.582,E2 -30314.582} C_VEL
LIN {X 0,Y 31.548,Z 494.949,A -85,B 0,C 180,E1 -30326.828,E2 -30326.828} C_VEL
LIN {X 0,Y 31.429,Z 486.284,A -85,B 0,C 180,E1 -30342.941,E2 -30342.941} C_VEL
LIN {X 0,Y 33.238,Z 476.78,A -85,B 0,C 180,E1 -30356.713,E2 -30356.713} C_VEL
LIN {X 0,Y 36.785,Z 464.84,A -85,B 0,C 180,E1 -30368.594,E2 -30368.594} C_VEL
LIN {X 0,Y 40.269,Z 453.262,A -85,B 0,C 180,E1 -30376.064,E2 -30376.064} C_VEL
LIN {X 0,Y 43.756,Z 440.162,A -85,B 0,C 180,E1 -30381.553,E2 -30381.553} C_VEL
LIN {X 0,Y 46.186,Z 427.891,A -85,B 0,C 180,E1 -30384.891,E2 -30384.891} C_VEL
LIN {X 0,Y 50.879,Z 395.754,A -85,B 0,C 180,E1 -30390.269,E2 -30390.269} C_VEL
LIN {X 0,Y 50.979,Z 384.449,A -85,B 0,C 180,E1 -30393.168,E2 -30393.168} C_VEL
LIN {X 0,Y 48.302,Z 370.324,A -85,B 0,C 180,E1 -30399.69,E2 -30399.69} C_VEL
LIN {X 0,Y 45.204,Z 361.366,A -85,B 0,C 180,E1 -30406.438,E2 -30406.438} C_VEL
LIN {X 0,Y 41.997,Z 353.775,A -85,B 0,C 180,E1 -30414.798,E2 -30414.798} C_VEL
LIN {X 0,Y 40.522,Z 350.732,A -85,B 0,C 180,E1 -30419.621,E2 -30419.621} C_VEL
LIN {X 0,Y 39.042,Z 347.682,A -85,B 0,C 180,E1 -30425.806,E2 -30425.806} C_VEL
LIN {X 0,Y 36.423,Z 345.442,A -85,B 0,C 180,E1 -30440.209,E2 -30440.209} C_VEL
LIN {X 0,Y 35.92,Z 344.806,A -85,B 0,C 180,E1 -30449.278,E2 -30449.278} C_VEL
LIN {X 0,Y 36.045,Z 345.178,A -85,B 0,C 180,E1 -30458.135,E2 -30458.135} C_VEL
LIN {X 0,Y 38.755,Z 348.394,A -85,B 0,C 180,E1 -30477.307,E2 -30477.307} C_VEL
LIN {X 0,Y 40.778,Z 351.695,A -85,B 0,C 180,E1 -30484.84,E2 -30484.84} C_VEL
LIN {X 0,Y 41.802,Z 353.148,A -85,B 0,C 180,E1 -30487.877,E2 -30487.877} C_VEL
LIN {X 0,Y 44.555,Z 357.803,A -85,B 0,C 180,E1 -30494.766,E2 -30494.766} C_VEL
LIN {X 0,Y 47.041,Z 365.291,A -85,B 0,C 180,E1 -30500.716,E2 -30500.716} C_VEL
LIN {X 0,Y 50.683,Z 378.227,A -85,B 0,C 180,E1 -30508.28,E2 -30508.28} C_VEL
LIN {X 0,Y 51.926,Z 382.93,A -85,B 0,C 180,E1 -30510.586,E2 -30510.586} C_VEL
LIN {X 0,Y 46.018,Z 422.947,A -85,B 0,C 180,E1 -30517.002,E2 -30517.002} C_VEL
LIN {X 0,Y 44.293,Z 428.579,A -85,B 0,C 180,E1 -30517.722,E2 -30517.722} C_VEL
LIN {X 0,Y 39.629,Z 437.341,A -85,B 0,C 180,E1 -30518.396,E2 -30518.396} C_VEL
LIN {X 0,Y 34.569,Z 445.862,A -85,B 0,C 180,E1 -30520.131,E2 -30520.131} C_VEL
LIN {X 0,Y 32.285,Z 451.127,A -85,B 0,C 180,E1 -30522.79,E2 -30522.79} C_VEL
LIN {X 0,Y 28.365,Z 462.346,A -85,B 0,C 180,E1 -30531.72,E2 -30531.72} C_VEL
LIN {X 0,Y 24.616,Z 473.984,A -85,B 0,C 180,E1 -30546.796,E2 -30546.796} C_VEL
LIN {X 0,Y 22.637,Z 484.38,A -85,B 0,C 180,E1 -30567.629,E2 -30567.629} C_VEL
LIN {X 0,Y 23.206,Z 491.76,A -85,B 0,C 180,E1 -30586.88,E2 -30586.88} C_VEL
LIN {X 0,Y 27.788,Z 500.914,A -85,B 0,C 180,E1 -30610.942,E2 -30610.942} C_VEL
LIN {X 0,Y 36.942,Z 509.42,A -85,B 0,C 180,E1 -30628.223,E2 -30628.223} C_VEL
LIN {X 0,Y 38.757,Z 510.717,A -85,B 0,C 180,E1 -30630.305,E2 -30630.305} C_VEL
LIN {X 0,Y 30.901,Z 504.874,A -85,B 0,C 180,E1 -30647.01,E2 -30647.01} C_VEL
LIN {X 0,Y 27.196,Z 498.747,A -85,B 0,C 180,E1 -30667.221,E2 -30667.221} C_VEL
LIN {X 0,Y 25.598,Z 494.513,A -85,B 0,C 180,E1 -30678.144,E2 -30678.144} C_VEL
LIN {X 0,Y 24.495,Z 485.888,A -85,B 0,C 180,E1 -30698.274,E2 -30698.274} C_VEL
LIN {X 0,Y 26.043,Z 476.467,A -85,B 0,C 180,E1 -30716.035,E2 -30716.035} C_VEL
LIN {X 0,Y 29.649,Z 464.866,A -85,B 0,C 180,E1 -30730.706,E2 -30730.706} C_VEL
LIN {X 0,Y 33.779,Z 452.348,A -85,B 0,C 180,E1 -30740.245,E2 -30740.245} C_VEL
LIN {X 0,Y 37.591,Z 439.14,A -85,B 0,C 180,E1 -30746.324,E2 -30746.324} C_VEL
LIN {X 0,Y 40.231,Z 426.626,A -85,B 0,C 180,E1 -30749.843,E2 -30749.843} C_VEL
LIN {X 0,Y 45.09,Z 395.29,A -85,B 0,C 180,E1 -30755.324,E2 -30755.324} C_VEL
LIN {X 0,Y 45.318,Z 385.944,A -85,B 0,C 180,E1 -30758.049,E2 -30758.049} C_VEL
LIN {X 0,Y 43.258,Z 373.29,A -85,B 0,C 180,E1 -30764.8,E2 -30764.8} C_VEL
LIN {X 0,Y 40.807,Z 365.186,A -85,B 0,C 180,E1 -30771.905,E2 -30771.905} C_VEL
LIN {X 0,Y 38.386,Z 358.286,A -85,B 0,C 180,E1 -30780.896,E2 -30780.896} C_VEL
LIN {X 0,Y 37.36,Z 355.815,A -85,B 0,C 180,E1 -30785.73,E2 -30785.73} C_VEL
LIN {X 0,Y 36.78,Z 354.266,A -85,B 0,C 180,E1 -30788.926,E2 -30788.926} C_VEL
LIN {X 0,Y 34.753,Z 352.207,A -85,B 0,C 180,E1 -30803.85,E2 -30803.85} C_VEL
LIN {X 0,Y 34.561,Z 351.816,A -85,B 0,C 180,E1 -30810.549,E2 -30810.549} C_VEL
LIN {X 0,Y 34.647,Z 352.266,A -85,B 0,C 180,E1 -30817.477,E2 -30817.477} C_VEL
LIN {X 0,Y 36.434,Z 354.813,A -85,B 0,C 180,E1 -30833.705,E2 -30833.705} C_VEL
LIN {X 0,Y 38.799,Z 359.01,A -85,B 0,C 180,E1 -30843.916,E2 -30843.916} C_VEL
LIN {X 0,Y 40.672,Z 362.646,A -85,B 0,C 180,E1 -30850.055,E2 -30850.055} C_VEL
LIN {X 0,Y 42.583,Z 369.784,A -85,B 0,C 180,E1 -30856.372,E2 -30856.372} C_VEL
LIN {X 0,Y 45.726,Z 382.712,A -85,B 0,C 180,E1 -30864.792,E2 -30864.792} C_VEL
LIN {X 0,Y 46.109,Z 384.476,A -85,B 0,C 180,E1 -30865.736,E2 -30865.736} C_VEL
LIN {X 0,Y 39.565,Z 424.525,A -85,B 0,C 180,E1 -30872.431,E2 -30872.431} C_VEL
LIN {X 0,Y 36.658,Z 436.923,A -85,B 0,C 180,E1 -30876.039,E2 -30876.039} C_VEL
LIN {X 0,Y 32.431,Z 450.677,A -85,B 0,C 180,E1 -30882.494,E2 -30882.494} C_VEL
LIN {X 0,Y 32.285,Z 451.127,A -85,B 0,C 180,E1 -30882.79,E2 -30882.79} C_VEL
LIN {X 0,Y 29.939,Z 456.25,A -85,B 0,C 180,E1 -30885.942,E2 -30885.942} C_VEL
LIN {X 0,Y 24.372,Z 464.006,A -85,B 0,C 180,E1 -30891.668,E2 -30891.668} C_VEL
LIN {X 0,Y 18.764,Z 471.414,A -85,B 0,C 180,E1 -30901.761,E2 -30901.761} C_VEL
LIN {X 0,Y 16.751,Z 475.985,A -85,B 0,C 180,E1 -30912.33,E2 -30912.33} C_VEL
LIN {X 0,Y 16.167,Z 485.773,A -85,B 0,C 180,E1 -30942.836,E2 -30942.836} C_VEL
LIN {X 0,Y 19.575,Z 494.14,A -85,B 0,C 180,E1 -30970.352,E2 -30970.352} C_VEL
LIN {X 0,Y 25.58,Z 501.01,A -85,B 0,C 180,E1 -30987.222,E2 -30987.222} C_VEL
LIN {X 0,Y 27.572,Z 502.726,A -85,B 0,C 180,E1 -30990.659,E2 -30990.659} C_VEL
LIN {X 0,Y 26.551,Z 501.94,A -85,B 0,C 180,E1 -30997.476,E2 -30997.476} C_VEL
LIN {X 0,Y 22.096,Z 496.646,A -85,B 0,C 180,E1 -31016.218,E2 -31016.218} C_VEL
LIN {X 0,Y 20.578,Z 493.982,A -85,B 0,C 180,E1 -31024.765,E2 -31024.765} C_VEL
LIN {X 0,Y 17.886,Z 485.515,A -85,B 0,C 180,E1 -31050.036,E2 -31050.036} C_VEL
LIN {X 0,Y 18.832,Z 476.137,A -85,B 0,C 180,E1 -31074.86,E2 -31074.86} C_VEL
LIN {X 0,Y 22.643,Z 464.588,A -85,B 0,C 180,E1 -31094.329,E2 -31094.329} C_VEL
LIN {X 0,Y 27.272,Z 452.022,A -85,B 0,C 180,E1 -31105.703,E2 -31105.703} C_VEL
LIN {X 0,Y 31.261,Z 439.612,A -85,B 0,C 180,E1 -31111.961,E2 -31111.961} C_VEL
LIN {X 0,Y 34.167,Z 427.457,A -85,B 0,C 180,E1 -31115.738,E2 -31115.738} C_VEL
LIN {X 0,Y 39.612,Z 395.392,A -85,B 0,C 180,E1 -31121.487,E2 -31121.487} C_VEL
LIN {X 0,Y 39.952,Z 387.571,A -85,B 0,C 180,E1 -31124.036,E2 -31124.036} C_VEL
LIN {X 0,Y 38.629,Z 376.442,A -85,B 0,C 180,E1 -31130.889,E2 -31130.889} C_VEL
LIN {X 0,Y 36.843,Z 368.873,A -85,B 0,C 180,E1 -31138.766,E2 -31138.766} C_VEL
LIN {X 0,Y 35.138,Z 362.427,A -85,B 0,C 180,E1 -31148.738,E2 -31148.738} C_VEL
LIN {X 0,Y 34.36,Z 360.51,A -85,B 0,C 180,E1 -31154.169,E2 -31154.169} C_VEL
LIN {X 0,Y 33.272,Z 359.021,A -85,B 0,C 180,E1 -31166.664,E2 -31166.664} C_VEL
LIN {X 0,Y 33.25,Z 358.992,A -85,B 0,C 180,E1 -31174.607,E2 -31174.607} C_VEL
LIN {X 0,Y 34.315,Z 361.291,A -85,B 0,C 180,E1 -31189.903,E2 -31189.903} C_VEL
LIN {X 0,Y 36.056,Z 365.159,A -85,B 0,C 180,E1 -31200.061,E2 -31200.061} C_VEL
LIN {X 0,Y 37.098,Z 367.637,A -85,B 0,C 180,E1 -31204.47,E2 -31204.47} C_VEL
LIN {X 0,Y 38.331,Z 373.826,A -85,B 0,C 180,E1 -31210.647,E2 -31210.647} C_VEL
LIN {X 0,Y 40.607,Z 385.798,A -85,B 0,C 180,E1 -31219.655,E2 -31219.655} C_VEL
LIN {X 0,Y 33.892,Z 423.912,A -85,B 0,C 180,E1 -31225.833,E2 -31225.833} C_VEL
LIN {X 0,Y 30.819,Z 436.228,A -85,B 0,C 180,E1 -31229.271,E2 -31229.271} C_VEL
LIN {X 0,Y 26.065,Z 450.464,A -85,B 0,C 180,E1 -31236.203,E2 -31236.203} C_VEL
LIN {X 0,Y 21.225,Z 462.901,A -85,B 0,C 180,E1 -31247.733,E2 -31247.733} C_VEL
LIN {X 0,Y 17.434,Z 473.503,A -85,B 0,C 180,E1 -31266.288,E2 -31266.288} C_VEL
LIN {X 0,Y 16.751,Z 475.985,A -85,B 0,C 180,E1 -31272.33,E2 -31272.33} C_VEL
LIN {X 0,Y 15.496,Z 478.858,A -85,B 0,C 180,E1 -31280.888,E2 -31280.888} C_VEL
LIN {X 0,Y 12.697,Z 482.763,A -85,B 0,C 180,E1 -31300.059,E2 -31300.059} C_VEL
LIN {X 0,Y 11.877,Z 486.443,A -85,B 0,C 180,E1 -31326.739,E2 -31326.739} C_VEL
LIN {X 0,Y 13.249,Z 488.992,A -85,B 0,C 180,E1 -31339.568,E2 -31339.568} C_VEL
LIN {X 0,Y 16.202,Z 492.476,A -85,B 0,C 180,E1 -31349.914,E2 -31349.914} C_VEL
LIN {X 0,Y 18.245,Z 494.462,A -85,B 0,C 180,E1 -31359.672,E2 -31359.672} C_VEL
LIN {X 0,Y 16.05,Z 491.765,A -85,B 0,C 180,E1 -31369,E2 -31369} C_VEL
LIN {X 0,Y 11.533,Z 482.993,A -85,B 0,C 180,E1 -31401.294,E2 -31401.294} C_VEL
LIN {X 0,Y 12.266,Z 473.368,A -85,B 0,C 180,E1 -31440.145,E2 -31440.145} C_VEL
LIN {X 0,Y 17.109,Z 461.346,A -85,B 0,C 180,E1 -31465.296,E2 -31465.296} C_VEL
LIN {X 0,Y 22.497,Z 448.268,A -85,B 0,C 180,E1 -31476.648,E2 -31476.648} C_VEL
LIN {X 0,Y 26.87,Z 435.016,A -85,B 0,C 180,E1 -31482.107,E2 -31482.107} C_VEL
LIN {X 0,Y 29.956,Z 421.543,A -85,B 0,C 180,E1 -31485.322,E2 -31485.322} C_VEL
LIN {X 0,Y 34.629,Z 395.959,A -85,B 0,C 180,E1 -31489.253,E2 -31489.253} C_VEL
LIN {X 0,Y 35.092,Z 389.164,A -85,B 0,C 180,E1 -31491.771,E2 -31491.771} C_VEL
LIN {X 0,Y 34.502,Z 379.553,A -85,B 0,C 180,E1 -31498.682,E2 -31498.682} C_VEL
LIN {X 0,Y 33.546,Z 373.284,A -85,B 0,C 180,E1 -31506.141,E2 -31506.141} C_VEL
LIN {X 0,Y 32.677,Z 367.859,A -85,B 0,C 180,E1 -31515.436,E2 -31515.436} C_VEL
LIN {X 0,Y 32.401,Z 366.994,A -85,B 0,C 180,E1 -31518.601,E2 -31518.601} C_VEL
LIN {X 0,Y 31.895,Z 365.908,A -85,B 0,C 180,E1 -31528.159,E2 -31528.159} C_VEL
LIN {X 0,Y 31.867,Z 365.924,A -85,B 0,C 180,E1 -31532.639,E2 -31532.639} C_VEL
LIN {X 0,Y 32.369,Z 367.74,A -85,B 0,C 180,E1 -31545.621,E2 -31545.621} C_VEL
LIN {X 0,Y 33.498,Z 371.251,A -85,B 0,C 180,E1 -31555.576,E2 -31555.576} C_VEL
LIN {X 0,Y 33.861,Z 372.932,A -85,B 0,C 180,E1 -31558.297,E2 -31558.297} C_VEL
LIN {X 0,Y 34.758,Z 380.012,A -85,B 0,C 180,E1 -31565.639,E2 -31565.639} C_VEL
LIN {X 0,Y 35.641,Z 387.387,A -85,B 0,C 180,E1 -31571.803,E2 -31571.803} C_VEL
LIN {X 0,Y 28.877,Z 423.065,A -85,B 0,C 180,E1 -31576.752,E2 -31576.752} C_VEL
LIN {X 0,Y 25.438,Z 435.9,A -85,B 0,C 180,E1 -31579.768,E2 -31579.768} C_VEL
LIN {X 0,Y 20.599,Z 449.001,A -85,B 0,C 180,E1 -31585.521,E2 -31585.521} C_VEL
LIN {X 0,Y 14.869,Z 461.943,A -85,B 0,C 180,E1 -31598.042,E2 -31598.042} C_VEL
LIN {X 0,Y 10.05,Z 473.64,A -85,B 0,C 180,E1 -31628.15,E2 -31628.15} C_VEL
LIN {X 0,Y 9.781,Z 482.252,A -85,B 0,C 180,E1 -31670.495,E2 -31670.495} C_VEL
LIN {X 0,Y 13.249,Z 488.992,A -85,B 0,C 180,E1 -31699.568,E2 -31699.568} C_VEL
LIN {X 0,Y 13.096,Z 489.077,A -85,B 0,C 180,E1 -31704.139,E2 -31704.139} C_VEL
LIN {X 0,Y 11.733,Z 487.773,A -85,B 0,C 180,E1 -31712.079,E2 -31712.079} C_VEL
LIN {X 0,Y 9.907,Z 485.603,A -85,B 0,C 180,E1 -31719.992,E2 -31719.992} C_VEL
LIN {X 0,Y 5.913,Z 479.696,A -85,B 0,C 180,E1 -31743.387,E2 -31743.387} C_VEL
LIN {X 0,Y 4.892,Z 473.471,A -85,B 0,C 180,E1 -31795.46,E2 -31795.46} C_VEL
LIN {X 0,Y 10.329,Z 462.24,A -85,B 0,C 180,E1 -31839.485,E2 -31839.485} C_VEL
LIN {X 0,Y 16.084,Z 450.647,A -85,B 0,C 180,E1 -31849.658,E2 -31849.658} C_VEL
LIN {X 0,Y 21.212,Z 437.779,A -85,B 0,C 180,E1 -31853.94,E2 -31853.94} C_VEL
LIN {X 0,Y 24.655,Z 425.28,A -85,B 0,C 180,E1 -31856.419,E2 -31856.419} C_VEL
LIN {X 0,Y 30.523,Z 396.085,A -85,B 0,C 180,E1 -31859.542,E2 -31859.542} C_VEL
LIN {X 0,Y 31.081,Z 390.583,A -85,B 0,C 180,E1 -31861.703,E2 -31861.703} C_VEL
LIN {X 0,Y 31.081,Z 382.611,A -85,B 0,C 180,E1 -31868.189,E2 -31868.189} C_VEL
LIN {X 0,Y 30.781,Z 377.037,A -85,B 0,C 180,E1 -31875.91,E2 -31875.91} C_VEL
LIN {X 0,Y 30.741,Z 373.687,A -85,B 0,C 180,E1 -31882.001,E2 -31882.001} C_VEL
LIN {X 0,Y 30.537,Z 372.837,A -85,B 0,C 180,E1 -31889.573,E2 -31889.573} C_VEL
LIN {X 0,Y 30.641,Z 374.201,A -85,B 0,C 180,E1 -31901.039,E2 -31901.039} C_VEL
LIN {X 0,Y 31.064,Z 376.832,A -85,B 0,C 180,E1 -31909.081,E2 -31909.081} C_VEL
LIN {X 0,Y 31.358,Z 385.742,A -85,B 0,C 180,E1 -31919.149,E2 -31919.149} C_VEL
LIN {X 0,Y 31.504,Z 388.575,A -85,B 0,C 180,E1 -31921.817,E2 -31921.817} C_VEL
LIN {X 0,Y 24.424,Z 423.315,A -85,B 0,C 180,E1 -31924.645,E2 -31924.645} C_VEL
LIN {X 0,Y 20.934,Z 435.574,A -85,B 0,C 180,E1 -31926.045,E2 -31926.045} C_VEL
LIN {X 0,Y 15.79,Z 448.571,A -85,B 0,C 180,E1 -31928.891,E2 -31928.891} C_VEL
LIN {X 0,Y 9.008,Z 461.82,A -85,B 0,C 180,E1 -31937.124,E2 -31937.124} C_VEL
LIN {X 0,Y 3.317,Z 471.876,A -85,B 0,C 180,E1 -31974.651,E2 -31974.651} C_VEL
LIN {X 0,Y 6.032,Z 480.932,A -85,B 0,C 180,E1 -32075.671,E2 -32075.671} C_VEL
LIN {X 0,Y 6.065,Z 480.409,A -85,B 0,C 180,E1 -32094.729,E2 -32094.729} C_VEL
LIN {X 0,Y 4.892,Z 473.471,A -85,B 0,C 180,E1 -32155.46,E2 -32155.46} C_VEL
LIN {X 0,Y 5.823,Z 470.251,A -85,B 0,C 180,E1 -32177.83,E2 -32177.83} C_VEL
LIN {X 0,Y 7.361,Z 465.176,A -85,B 0,C 180,E1 -32201.388,E2 -32201.388} C_VEL
LIN {X 0,Y 11.786,Z 452.769,A -85,B 0,C 180,E1 -32230.906,E2 -32230.906} C_VEL
LIN {X 0,Y 14.022,Z 447.307,A -85,B 0,C 180,E1 -32233.904,E2 -32233.904} C_VEL
LIN {X 0,Y 14.797,Z 445.435,A -85,B 0,C 180,E1 -32233.648,E2 -32233.648} C_VEL
LIN {X 0,Y 19.558,Z 432.339,A -85,B 0,C 180,E1 -32232.19,E2 -32232.19} C_VEL
LIN {X 0,Y 23.402,Z 416.23,A -85,B 0,C 180,E1 -32232.016,E2 -32232.016} C_VEL
LIN {X 0,Y 27.568,Z 395.558,A -85,B 0,C 180,E1 -32232.476,E2 -32232.476} C_VEL
LIN {X 0,Y 28.047,Z 392.016,A -85,B 0,C 180,E1 -32234.042,E2 -32234.042} C_VEL
LIN {X 0,Y 28.657,Z 385.262,A -85,B 0,C 180,E1 -32240.085,E2 -32240.085} C_VEL
LIN {X 0,Y 29.155,Z 380.162,A -85,B 0,C 180,E1 -32248.307,E2 -32248.307} C_VEL
LIN {X 0,Y 29.143,Z 380.056,A -85,B 0,C 180,E1 -32251.14,E2 -32251.14} C_VEL
LIN {X 0,Y 29.108,Z 380.884,A -85,B 0,C 180,E1 -32256.575,E2 -32256.575} C_VEL
LIN {X 0,Y 29.067,Z 382.023,A -85,B 0,C 180,E1 -32260.184,E2 -32260.184} C_VEL
LIN {X 0,Y 28.453,Z 390.038,A -85,B 0,C 180,E1 -32269.377,E2 -32269.377} C_VEL
LIN {X 0,Y 21.147,Z 425.09,A -85,B 0,C 180,E1 -32268.306,E2 -32268.306} C_VEL
LIN {X 0,Y 17.111,Z 438.334,A -85,B 0,C 180,E1 -32265.936,E2 -32265.936} C_VEL
LIN {X 0,Y 12.11,Z 450.562,A -85,B 0,C 180,E1 -32260.738,E2 -32260.738} C_VEL
LIN {X 0,Y 8.312,Z 458.346,A -85,B 0,C 180,E1 -32252.137,E2 -32252.137} C_VEL
LIN {X 0,Y 7.526,Z 460.126,A -85,B 0,C 180,E1 -32240.726,E2 -32240.726} C_VEL
LIN {X 0,Y 14.047,Z 447.218,A -85,B 0,C 180,E1 -32234.05,E2 -32234.05} C_VEL
LIN {X 0,Y 14.797,Z 445.435,A -85,B 0,C 180,E1 -32233.648,E2 -32233.648} C_VEL
LIN {X 0,Y 17.424,Z 438.419,A -85,B 0,C 180,E1 -32233.803,E2 -32233.803} C_VEL
LIN {X 0,Y 19.421,Z 431.16,A -85,B 0,C 180,E1 -32236.807,E2 -32236.807} C_VEL
LIN {X 0,Y 21.373,Z 421.375,A -85,B 0,C 180,E1 -32242.865,E2 -32242.865} C_VEL
LIN {X 0,Y 23.109,Z 411.481,A -85,B 0,C 180,E1 -32247.779,E2 -32247.779} C_VEL
LIN {X 0,Y 24.047,Z 406.484,A -85,B 0,C 180,E1 -32248.282,E2 -32248.282} C_VEL
LIN {X 0,Y 26.185,Z 395.595,A -85,B 0,C 180,E1 -32247.4,E2 -32247.4} C_VEL
LIN {X 0,Y 26.954,Z 391.388,A -85,B 0,C 180,E1 -32250.035,E2 -32250.035} C_VEL
LIN {X 0,Y 27.392,Z 389.143,A -85,B 0,C 180,E1 -32252.146,E2 -32252.146} C_VEL
LIN {X 0,Y 26.952,Z 391.679,A -85,B 0,C 180,E1 -32254.736,E2 -32254.736} C_VEL
LIN {X 0,Y 22.006,Z 416.856,A -85,B 0,C 180,E1 -32250.948,E2 -32250.948} C_VEL
LIN {X 0,Y 22,Z 416.917,A -85,B 0,C 180,E1 -32249.787,E2 -32249.787} C_VEL
LIN {X 0,Y 24.047,Z 406.484,A -85,B 0,C 180,E1 -32248.282,E2 -32248.282} C_VEL
LIN {X 0,Y 27.954,Z 406.875,A -85,B 0,C 180,E1 -32246.835,E2 -32246.835} C_VEL
LIN {X 0,Y 27.954,Z 600,A -85,B 0,C 180,E1 -32246.835,E2 -32246.835} C_VEL
LIN {X 0,Y 27.954,Z 600,A -85,B 0,C 180,E1 -32246.835,E2 -32246.835}

QRS_NEXT_CUT()

QRS_NEXT()
QRS_HOME()

END
